LIN {X 91.341,Y 104.941,Z 79.000,A 180.000,B 0.000,C 180.000} C_DIS
LIN {X 91.355,Y 104.953,Z 79.000,A 180.000,B 0.000,C 180.000} C_DIS
LIN {X 91.533,Y 105.100,Z 79.000,A 180.000,B 0.000,C 180.000} C_DIS
LIN {X 91.560,Y 105.120,Z 79.000,A 180.000,B 0.000,C 180.000} C_DIS
LIN {X 91.712,Y 105.235,Z 79.000,A 180.000,B 0.000,C 180.000} C_DIS
LIN {X 91.797,Y 105.299,Z 79.000,A 180.000,B 0.000,C 180.000} C_DIS
LIN {X 91.891,Y 105.368,Z 79.000,A 180.000,B 0.000,C 180.000} C_DIS
LIN {X 92.052,Y 105.477,Z 79.000,A 180.000,B 0.000,C 180.000} C_DIS
LIN {X 92.070,Y 105.489,Z 79.000,A 180.000,B 0.000,C 180.000} C_DIS
LIN {X 92.249,Y 105.609,Z 79.000,A 180.000,B 0.000,C 180.000} C_DIS
LIN {X 92.323,Y 105.656,Z 79.000,A 180.000,B 0.000,C 180.000} C_DIS
LIN {X 92.427,Y 105.722,Z 79.000,A 180.000,B 0.000,C 180.000} C_DIS
LIN {X 92.606,Y 105.829,Z 79.000,A 180.000,B 0.000,C 180.000} C_DIS
LIN {X 92.785,Y 105.934,Z 79.000,A 180.000,B 0.000,C 180.000} C_DIS
LIN {X 92.933,Y 106.014,Z 79.000,A 180.000,B 0.000,C 180.000} C_DIS
LIN {X 93.142,Y 106.122,Z 79.000,A 180.000,B 0.000,C 180.000} C_DIS
LIN {X 93.284,Y 106.193,Z 79.000,A 180.000,B 0.000,C 180.000} C_DIS
LIN {X 93.321,Y 106.210,Z 79.000,A 180.000,B 0.000,C 180.000} C_DIS
LIN {X 93.500,Y 106.293,Z 79.000,A 180.000,B 0.000,C 180.000} C_DIS
LIN {X 93.679,Y 106.373,Z 79.000,A 180.000,B 0.000,C 180.000} C_DIS
LIN {X 93.857,Y 106.450,Z 79.000,A 180.000,B 0.000,C 180.000} C_DIS
LIN {X 94.036,Y 106.518,Z 79.000,A 180.000,B 0.000,C 180.000} C_DIS
LIN {X 94.119,Y 106.550,Z 79.000,A 180.000,B 0.000,C 180.000} C_DIS
LIN {X 94.215,Y 106.587,Z 79.000,A 180.000,B 0.000,C 180.000} C_DIS
LIN {X 94.321,Y 106.622,Z 79.000,A 180.000,B 0.000,C 180.000} C_DIS
; Link Move Starts
LIN {X 94.610,Y 106.716,Z 79.000,A 180.000,B 0.000,C 180.000} C_DIS
LIN {X 94.889,Y 106.804,Z 78.999,A 180.000,B 0.000,C 180.000} C_DIS
LIN {X 95.191,Y 106.882,Z 78.998,A 180.000,B 0.000,C 180.000} C_DIS
LIN {X 95.473,Y 106.946,Z 78.996,A 180.000,B 0.000,C 180.000} C_DIS
LIN {X 95.778,Y 107.008,Z 78.994,A 180.000,B 0.000,C 180.000} C_DIS
LIN {X 96.070,Y 107.058,Z 78.992,A 180.000,B 0.000,C 180.000} C_DIS
LIN {X 96.375,Y 107.102,Z 78.989,A 180.000,B 0.000,C 180.000} C_DIS
LIN {X 96.666,Y 107.130,Z 78.986,A 180.000,B 0.000,C 180.000} C_DIS
LIN {X 96.966,Y 107.154,Z 78.983,A 180.000,B 0.000,C 180.000} C_DIS
LIN {X 97.269,Y 107.168,Z 78.979,A 180.000,B 0.000,C 180.000} C_DIS
LIN {X 97.568,Y 107.174,Z 78.974,A 180.000,B 0.000,C 180.000} C_DIS
LIN {X 97.873,Y 107.168,Z 78.970,A 180.000,B 0.000,C 180.000} C_DIS
LIN {X 98.166,Y 107.154,Z 78.965,A 180.000,B 0.000,C 180.000} C_DIS
LIN {X 98.319,Y 107.143,Z 78.962,A 180.000,B 0.000,C 180.000} C_DIS
LIN {X 98.472,Y 107.131,Z 78.959,A 180.000,B 0.000,C 180.000} C_DIS
LIN {X 98.619,Y 107.118,Z 78.956,A 180.000,B 0.000,C 180.000} C_DIS
LIN {X 98.766,Y 107.100,Z 78.953,A 180.000,B 0.000,C 180.000} C_DIS
LIN {X 98.917,Y 107.080,Z 78.950,A 180.000,B 0.000,C 180.000} C_DIS
LIN {X 99.068,Y 107.059,Z 78.947,A 180.000,B 0.000,C 180.000} C_DIS
LIN {X 99.216,Y 107.033,Z 78.944,A 180.000,B 0.000,C 180.000} C_DIS
LIN {X 99.364,Y 107.005,Z 78.941,A 180.000,B 0.000,C 180.000} C_DIS
LIN {X 99.513,Y 106.977,Z 78.937,A 180.000,B 0.000,C 180.000} C_DIS
LIN {X 99.662,Y 106.949,Z 78.934,A 180.000,B 0.000,C 180.000} C_DIS
LIN {X 99.809,Y 106.915,Z 78.930,A 180.000,B 0.000,C 180.000} C_DIS
LIN {X 99.956,Y 106.879,Z 78.927,A 180.000,B 0.000,C 180.000} C_DIS
LIN {X 100.097,Y 106.844,Z 78.923,A 180.000,B 0.000,C 180.000} C_DIS
LIN {X 100.238,Y 106.804,Z 78.920,A 180.000,B 0.000,C 180.000} C_DIS
LIN {X 100.387,Y 106.758,Z 78.916,A 180.000,B 0.000,C 180.000} C_DIS
LIN {X 100.537,Y 106.713,Z 78.912,A 180.000,B 0.000,C 180.000} C_DIS
LIN {X 100.680,Y 106.668,Z 78.908,A 180.000,B 0.000,C 180.000} C_DIS
LIN {X 100.823,Y 106.620,Z 78.904,A 180.000,B 0.000,C 180.000} C_DIS
LIN {X 100.965,Y 106.568,Z 78.900,A 180.000,B 0.000,C 180.000} C_DIS
LIN {X 101.108,Y 106.516,Z 78.896,A 180.000,B 0.000,C 180.000} C_DIS
LIN {X 101.245,Y 106.462,Z 78.891,A 180.000,B 0.000,C 180.000} C_DIS
LIN {X 101.381,Y 106.403,Z 78.887,A 180.000,B 0.000,C 180.000} C_DIS
LIN {X 101.523,Y 106.342,Z 78.883,A 180.000,B 0.000,C 180.000} C_DIS
LIN {X 101.665,Y 106.279,Z 78.878,A 180.000,B 0.000,C 180.000} C_DIS
LIN {X 101.800,Y 106.218,Z 78.874,A 180.000,B 0.000,C 180.000} C_DIS
LIN {X 101.934,Y 106.151,Z 78.869,A 180.000,B 0.000,C 180.000} C_DIS
LIN {X 102.068,Y 106.084,Z 78.864,A 180.000,B 0.000,C 180.000} C_DIS
LIN {X 102.203,Y 106.016,Z 78.860,A 180.000,B 0.000,C 180.000} C_DIS
LIN {X 102.336,Y 105.941,Z 78.855,A 180.000,B 0.000,C 180.000} C_DIS
LIN {X 102.470,Y 105.865,Z 78.850,A 180.000,B 0.000,C 180.000} C_DIS
LIN {X 102.601,Y 105.790,Z 78.845,A 180.000,B 0.000,C 180.000} C_DIS
LIN {X 102.730,Y 105.711,Z 78.840,A 180.000,B 0.000,C 180.000} C_DIS
LIN {X 102.795,Y 105.671,Z 78.838,A 180.000,B 0.000,C 180.000} C_DIS
LIN {X 102.859,Y 105.629,Z 78.835,A 180.000,B 0.000,C 180.000} C_DIS
LIN {X 102.923,Y 105.588,Z 78.833,A 180.000,B 0.000,C 180.000} C_DIS
LIN {X 102.987,Y 105.546,Z 78.830,A 180.000,B 0.000,C 180.000} C_DIS
LIN {X 103.050,Y 105.506,Z 78.828,A 180.000,B 0.000,C 180.000} C_DIS
LIN {X 103.113,Y 105.465,Z 78.825,A 180.000,B 0.000,C 180.000} C_DIS
LIN {X 103.174,Y 105.423,Z 78.823,A 180.000,B 0.000,C 180.000} C_DIS
LIN {X 103.235,Y 105.380,Z 78.820,A 180.000,B 0.000,C 180.000} C_DIS
LIN {X 103.298,Y 105.334,Z 78.817,A 180.000,B 0.000,C 180.000} C_DIS
LIN {X 103.422,Y 105.243,Z 78.812,A 180.000,B 0.000,C 180.000} C_DIS
LIN {X 103.485,Y 105.198,Z 78.809,A 180.000,B 0.000,C 180.000} C_DIS
LIN {X 103.544,Y 105.153,Z 78.807,A 180.000,B 0.000,C 180.000} C_DIS
LIN {X 103.602,Y 105.107,Z 78.804,A 180.000,B 0.000,C 180.000} C_DIS
LIN {X 103.659,Y 105.061,Z 78.802,A 180.000,B 0.000,C 180.000} C_DIS
LIN {X 103.717,Y 105.015,Z 78.799,A 180.000,B 0.000,C 180.000} C_DIS
LIN {X 103.839,Y 104.915,Z 78.793,A 180.000,B 0.000,C 180.000} C_DIS
LIN {X 103.960,Y 104.816,Z 78.788,A 180.000,B 0.000,C 180.000} C_DIS
LIN {X 104.017,Y 104.769,Z 78.785,A 180.000,B 0.000,C 180.000} C_DIS
LIN {X 104.073,Y 104.720,Z 78.783,A 180.000,B 0.000,C 180.000} C_DIS
LIN {X 104.127,Y 104.671,Z 78.780,A 180.000,B 0.000,C 180.000} C_DIS
LIN {X 104.181,Y 104.621,Z 78.778,A 180.000,B 0.000,C 180.000} C_DIS
LIN {X 104.293,Y 104.519,Z 78.772,A 180.000,B 0.000,C 180.000} C_DIS
LIN {X 104.348,Y 104.468,Z 78.770,A 180.000,B 0.000,C 180.000} C_DIS
LIN {X 104.402,Y 104.416,Z 78.767,A 180.000,B 0.000,C 180.000} C_DIS
LIN {X 104.456,Y 104.361,Z 78.764,A 180.000,B 0.000,C 180.000} C_DIS
LIN {X 104.564,Y 104.250,Z 78.759,A 180.000,B 0.000,C 180.000} C_DIS
LIN {X 104.618,Y 104.195,Z 78.756,A 180.000,B 0.000,C 180.000} C_DIS
LIN {X 104.671,Y 104.141,Z 78.754,A 180.000,B 0.000,C 180.000} C_DIS
LIN {X 104.776,Y 104.032,Z 78.748,A 180.000,B 0.000,C 180.000} C_DIS
LIN {X 104.828,Y 103.978,Z 78.746,A 180.000,B 0.000,C 180.000} C_DIS
LIN {X 104.880,Y 103.920,Z 78.743,A 180.000,B 0.000,C 180.000} C_DIS
LIN {X 104.981,Y 103.804,Z 78.738,A 180.000,B 0.000,C 180.000} C_DIS
LIN {X 105.032,Y 103.746,Z 78.735,A 180.000,B 0.000,C 180.000} C_DIS
LIN {X 105.080,Y 103.690,Z 78.732,A 180.000,B 0.000,C 180.000} C_DIS
LIN {X 105.129,Y 103.634,Z 78.730,A 180.000,B 0.000,C 180.000} C_DIS
LIN {X 105.175,Y 103.577,Z 78.727,A 180.000,B 0.000,C 180.000} C_DIS
LIN {X 105.221,Y 103.518,Z 78.725,A 180.000,B 0.000,C 180.000} C_DIS
LIN {X 105.316,Y 103.396,Z 78.719,A 180.000,B 0.000,C 180.000} C_DIS
LIN {X 105.364,Y 103.334,Z 78.717,A 180.000,B 0.000,C 180.000} C_DIS
LIN {X 105.411,Y 103.273,Z 78.714,A 180.000,B 0.000,C 180.000} C_DIS
LIN {X 105.502,Y 103.153,Z 78.709,A 180.000,B 0.000,C 180.000} C_DIS
LIN {X 105.546,Y 103.092,Z 78.706,A 180.000,B 0.000,C 180.000} C_DIS
LIN {X 105.590,Y 103.030,Z 78.703,A 180.000,B 0.000,C 180.000} C_DIS
LIN {X 105.676,Y 102.905,Z 78.698,A 180.000,B 0.000,C 180.000} C_DIS
LIN {X 105.763,Y 102.779,Z 78.693,A 180.000,B 0.000,C 180.000} C_DIS
LIN {X 105.806,Y 102.715,Z 78.690,A 180.000,B 0.000,C 180.000} C_DIS
LIN {X 105.847,Y 102.650,Z 78.687,A 180.000,B 0.000,C 180.000} C_DIS
LIN {X 106.006,Y 102.389,Z 78.677,A 180.000,B 0.000,C 180.000} C_DIS
LIN {X 106.046,Y 102.324,Z 78.674,A 180.000,B 0.000,C 180.000} C_DIS
LIN {X 106.084,Y 102.257,Z 78.671,A 180.000,B 0.000,C 180.000} C_DIS
LIN {X 106.122,Y 102.191,Z 78.669,A 180.000,B 0.000,C 180.000} C_DIS
LIN {X 106.159,Y 102.124,Z 78.666,A 180.000,B 0.000,C 180.000} C_DIS
LIN {X 106.196,Y 102.056,Z 78.663,A 180.000,B 0.000,C 180.000} C_DIS
LIN {X 106.268,Y 101.922,Z 78.658,A 180.000,B 0.000,C 180.000} C_DIS
LIN {X 106.303,Y 101.856,Z 78.655,A 180.000,B 0.000,C 180.000} C_DIS
LIN {X 106.339,Y 101.790,Z 78.653,A 180.000,B 0.000,C 180.000} C_DIS
LIN {X 106.372,Y 101.723,Z 78.650,A 180.000,B 0.000,C 180.000} C_DIS
LIN {X 106.406,Y 101.652,Z 78.647,A 180.000,B 0.000,C 180.000} C_DIS
LIN {X 106.505,Y 101.440,Z 78.639,A 180.000,B 0.000,C 180.000} C_DIS
LIN {X 106.537,Y 101.371,Z 78.637,A 180.000,B 0.000,C 180.000} C_DIS
LIN {X 106.567,Y 101.302,Z 78.634,A 180.000,B 0.000,C 180.000} C_DIS
LIN {X 106.597,Y 101.232,Z 78.631,A 180.000,B 0.000,C 180.000} C_DIS
LIN {X 106.625,Y 101.163,Z 78.629,A 180.000,B 0.000,C 180.000} C_DIS
LIN {X 106.655,Y 101.091,Z 78.626,A 180.000,B 0.000,C 180.000} C_DIS
LIN {X 106.769,Y 100.805,Z 78.615,A 180.000,B 0.000,C 180.000} C_DIS
LIN {X 106.797,Y 100.735,Z 78.613,A 180.000,B 0.000,C 180.000} C_DIS
LIN {X 106.822,Y 100.664,Z 78.610,A 180.000,B 0.000,C 180.000} C_DIS
LIN {X 106.846,Y 100.593,Z 78.607,A 180.000,B 0.000,C 180.000} C_DIS
LIN {X 106.920,Y 100.372,Z 78.599,A 180.000,B 0.000,C 180.000} C_DIS
LIN {X 106.945,Y 100.299,Z 78.596,A 180.000,B 0.000,C 180.000} C_DIS
LIN {X 106.967,Y 100.226,Z 78.594,A 180.000,B 0.000,C 180.000} C_DIS
LIN {X 106.987,Y 100.153,Z 78.591,A 180.000,B 0.000,C 180.000} C_DIS
LIN {X 107.048,Y 99.930,Z 78.583,A 180.000,B 0.000,C 180.000} C_DIS
LIN {X 107.069,Y 99.855,Z 78.580,A 180.000,B 0.000,C 180.000} C_DIS
LIN {X 107.090,Y 99.779,Z 78.578,A 180.000,B 0.000,C 180.000} C_DIS
LIN {X 107.111,Y 99.703,Z 78.575,A 180.000,B 0.000,C 180.000} C_DIS
LIN {X 107.129,Y 99.630,Z 78.572,A 180.000,B 0.000,C 180.000} C_DIS
LIN {X 107.145,Y 99.557,Z 78.570,A 180.000,B 0.000,C 180.000} C_DIS
LIN {X 107.209,Y 99.262,Z 78.559,A 180.000,B 0.000,C 180.000} C_DIS
LIN {X 107.224,Y 99.188,Z 78.556,A 180.000,B 0.000,C 180.000} C_DIS
LIN {X 107.237,Y 99.114,Z 78.554,A 180.000,B 0.000,C 180.000} C_DIS
LIN {X 107.286,Y 98.806,Z 78.543,A 180.000,B 0.000,C 180.000} C_DIS
LIN {X 107.298,Y 98.729,Z 78.540,A 180.000,B 0.000,C 180.000} C_DIS
LIN {X 107.320,Y 98.575,Z 78.535,A 180.000,B 0.000,C 180.000} C_DIS
LIN {X 107.329,Y 98.498,Z 78.532,A 180.000,B 0.000,C 180.000} C_DIS
LIN {X 107.337,Y 98.422,Z 78.529,A 180.000,B 0.000,C 180.000} C_DIS
LIN {X 107.360,Y 98.192,Z 78.521,A 180.000,B 0.000,C 180.000} C_DIS
LIN {X 107.368,Y 98.117,Z 78.519,A 180.000,B 0.000,C 180.000} C_DIS
LIN {X 107.374,Y 98.042,Z 78.516,A 180.000,B 0.000,C 180.000} C_DIS
LIN {X 107.378,Y 97.967,Z 78.513,A 180.000,B 0.000,C 180.000} C_DIS
LIN {X 107.391,Y 97.660,Z 78.503,A 180.000,B 0.000,C 180.000} C_DIS
LIN {X 107.394,Y 97.583,Z 78.500,A 180.000,B 0.000,C 180.000} C_DIS
LIN {X 107.396,Y 97.429,Z 78.495,A 180.000,B 0.000,C 180.000} C_DIS
LIN {X 107.397,Y 97.352,Z 78.492,A 180.000,B 0.000,C 180.000} C_DIS
LIN {X 107.393,Y 97.040,Z 78.481,A 180.000,B 0.000,C 180.000} C_DIS
LIN {X 107.392,Y 96.962,Z 78.478,A 180.000,B 0.000,C 180.000} C_DIS
LIN {X 107.388,Y 96.886,Z 78.476,A 180.000,B 0.000,C 180.000} C_DIS
LIN {X 107.383,Y 96.810,Z 78.473,A 180.000,B 0.000,C 180.000} C_DIS
LIN {X 107.368,Y 96.581,Z 78.465,A 180.000,B 0.000,C 180.000} C_DIS
LIN {X 107.362,Y 96.505,Z 78.462,A 180.000,B 0.000,C 180.000} C_DIS
LIN {X 107.355,Y 96.429,Z 78.460,A 180.000,B 0.000,C 180.000} C_DIS
LIN {X 107.347,Y 96.353,Z 78.457,A 180.000,B 0.000,C 180.000} C_DIS
LIN {X 107.339,Y 96.275,Z 78.454,A 180.000,B 0.000,C 180.000} C_DIS
LIN {X 107.329,Y 96.198,Z 78.452,A 180.000,B 0.000,C 180.000} C_DIS
LIN {X 107.291,Y 95.890,Z 78.441,A 180.000,B 0.000,C 180.000} C_DIS
LIN {X 107.281,Y 95.814,Z 78.438,A 180.000,B 0.000,C 180.000} C_DIS
LIN {X 107.268,Y 95.739,Z 78.435,A 180.000,B 0.000,C 180.000} C_DIS
LIN {X 107.212,Y 95.433,Z 78.425,A 180.000,B 0.000,C 180.000} C_DIS
LIN {X 107.198,Y 95.358,Z 78.422,A 180.000,B 0.000,C 180.000} C_DIS
LIN {X 107.182,Y 95.283,Z 78.419,A 180.000,B 0.000,C 180.000} C_DIS
LIN {X 107.164,Y 95.209,Z 78.417,A 180.000,B 0.000,C 180.000} C_DIS
LIN {X 107.147,Y 95.135,Z 78.414,A 180.000,B 0.000,C 180.000} C_DIS
LIN {X 107.128,Y 95.058,Z 78.411,A 180.000,B 0.000,C 180.000} C_DIS
LIN {X 107.073,Y 94.828,Z 78.403,A 180.000,B 0.000,C 180.000} C_DIS
LIN {X 107.055,Y 94.754,Z 78.400,A 180.000,B 0.000,C 180.000} C_DIS
LIN {X 107.035,Y 94.681,Z 78.398,A 180.000,B 0.000,C 180.000} C_DIS
LIN {X 107.014,Y 94.608,Z 78.395,A 180.000,B 0.000,C 180.000} C_DIS
LIN {X 106.970,Y 94.461,Z 78.390,A 180.000,B 0.000,C 180.000} C_DIS
LIN {X 106.925,Y 94.314,Z 78.384,A 180.000,B 0.000,C 180.000} C_DIS
LIN {X 106.902,Y 94.241,Z 78.381,A 180.000,B 0.000,C 180.000} C_DIS
LIN {X 106.877,Y 94.167,Z 78.379,A 180.000,B 0.000,C 180.000} C_DIS
LIN {X 106.770,Y 93.873,Z 78.368,A 180.000,B 0.000,C 180.000} C_DIS
LIN {X 106.743,Y 93.800,Z 78.365,A 180.000,B 0.000,C 180.000} C_DIS
LIN {X 106.716,Y 93.728,Z 78.362,A 180.000,B 0.000,C 180.000} C_DIS
LIN {X 106.688,Y 93.655,Z 78.360,A 180.000,B 0.000,C 180.000} C_DIS
LIN {X 106.659,Y 93.583,Z 78.357,A 180.000,B 0.000,C 180.000} C_DIS
LIN {X 106.629,Y 93.512,Z 78.354,A 180.000,B 0.000,C 180.000} C_DIS
LIN {X 106.538,Y 93.299,Z 78.346,A 180.000,B 0.000,C 180.000} C_DIS
LIN {X 106.507,Y 93.228,Z 78.343,A 180.000,B 0.000,C 180.000} C_DIS
LIN {X 106.475,Y 93.158,Z 78.341,A 180.000,B 0.000,C 180.000} C_DIS
LIN {X 106.441,Y 93.089,Z 78.338,A 180.000,B 0.000,C 180.000} C_DIS
LIN {X 106.372,Y 92.949,Z 78.333,A 180.000,B 0.000,C 180.000} C_DIS
LIN {X 106.303,Y 92.810,Z 78.327,A 180.000,B 0.000,C 180.000} C_DIS
LIN {X 106.267,Y 92.741,Z 78.325,A 180.000,B 0.000,C 180.000} C_DIS
LIN {X 106.231,Y 92.672,Z 78.322,A 180.000,B 0.000,C 180.000} C_DIS
LIN {X 106.194,Y 92.603,Z 78.319,A 180.000,B 0.000,C 180.000} C_DIS
LIN {X 106.157,Y 92.535,Z 78.316,A 180.000,B 0.000,C 180.000} C_DIS
LIN {X 106.080,Y 92.400,Z 78.311,A 180.000,B 0.000,C 180.000} C_DIS
LIN {X 106.003,Y 92.265,Z 78.306,A 180.000,B 0.000,C 180.000} C_DIS
LIN {X 105.965,Y 92.198,Z 78.303,A 180.000,B 0.000,C 180.000} C_DIS
LIN {X 105.924,Y 92.132,Z 78.300,A 180.000,B 0.000,C 180.000} C_DIS
LIN {X 105.882,Y 92.067,Z 78.297,A 180.000,B 0.000,C 180.000} C_DIS
LIN {X 105.840,Y 92.002,Z 78.295,A 180.000,B 0.000,C 180.000} C_DIS
LIN {X 105.756,Y 91.872,Z 78.289,A 180.000,B 0.000,C 180.000} C_DIS
LIN {X 105.714,Y 91.807,Z 78.287,A 180.000,B 0.000,C 180.000} C_DIS
LIN {X 105.670,Y 91.743,Z 78.284,A 180.000,B 0.000,C 180.000} C_DIS
LIN {X 105.581,Y 91.615,Z 78.278,A 180.000,B 0.000,C 180.000} C_DIS
LIN {X 105.535,Y 91.551,Z 78.276,A 180.000,B 0.000,C 180.000} C_DIS
LIN {X 105.489,Y 91.488,Z 78.273,A 180.000,B 0.000,C 180.000} C_DIS
LIN {X 105.398,Y 91.363,Z 78.268,A 180.000,B 0.000,C 180.000} C_DIS
LIN {X 105.353,Y 91.301,Z 78.265,A 180.000,B 0.000,C 180.000} C_DIS
LIN {X 105.306,Y 91.239,Z 78.262,A 180.000,B 0.000,C 180.000} C_DIS
LIN {X 105.257,Y 91.177,Z 78.259,A 180.000,B 0.000,C 180.000} C_DIS
LIN {X 105.158,Y 91.056,Z 78.254,A 180.000,B 0.000,C 180.000} C_DIS
LIN {X 105.108,Y 90.995,Z 78.251,A 180.000,B 0.000,C 180.000} C_DIS
LIN {X 105.059,Y 90.935,Z 78.249,A 180.000,B 0.000,C 180.000} C_DIS
LIN {X 105.009,Y 90.875,Z 78.246,A 180.000,B 0.000,C 180.000} C_DIS
LIN {X 104.958,Y 90.817,Z 78.243,A 180.000,B 0.000,C 180.000} C_DIS
LIN {X 104.906,Y 90.760,Z 78.240,A 180.000,B 0.000,C 180.000} C_DIS
LIN {X 104.853,Y 90.702,Z 78.238,A 180.000,B 0.000,C 180.000} C_DIS
LIN {X 104.800,Y 90.644,Z 78.235,A 180.000,B 0.000,C 180.000} C_DIS
LIN {X 104.642,Y 90.471,Z 78.227,A 180.000,B 0.000,C 180.000} C_DIS
LIN {X 104.590,Y 90.414,Z 78.224,A 180.000,B 0.000,C 180.000} C_DIS
LIN {X 104.536,Y 90.358,Z 78.221,A 180.000,B 0.000,C 180.000} C_DIS
LIN {X 104.481,Y 90.304,Z 78.219,A 180.000,B 0.000,C 180.000} C_DIS
LIN {X 104.369,Y 90.195,Z 78.213,A 180.000,B 0.000,C 180.000} C_DIS
LIN {X 104.257,Y 90.085,Z 78.208,A 180.000,B 0.000,C 180.000} C_DIS
LIN {X 104.200,Y 90.032,Z 78.205,A 180.000,B 0.000,C 180.000} C_DIS
LIN {X 104.142,Y 89.980,Z 78.202,A 180.000,B 0.000,C 180.000} C_DIS
LIN {X 103.966,Y 89.826,Z 78.194,A 180.000,B 0.000,C 180.000} C_DIS
LIN {X 103.906,Y 89.774,Z 78.191,A 180.000,B 0.000,C 180.000} C_DIS
LIN {X 103.847,Y 89.723,Z 78.189,A 180.000,B 0.000,C 180.000} C_DIS
LIN {X 103.787,Y 89.672,Z 78.186,A 180.000,B 0.000,C 180.000} C_DIS
LIN {X 103.728,Y 89.622,Z 78.183,A 180.000,B 0.000,C 180.000} C_DIS
LIN {X 103.667,Y 89.573,Z 78.181,A 180.000,B 0.000,C 180.000} C_DIS
LIN {X 103.606,Y 89.525,Z 78.178,A 180.000,B 0.000,C 180.000} C_DIS
LIN {X 103.483,Y 89.429,Z 78.173,A 180.000,B 0.000,C 180.000} C_DIS
LIN {X 103.421,Y 89.381,Z 78.170,A 180.000,B 0.000,C 180.000} C_DIS
LIN {X 103.358,Y 89.333,Z 78.167,A 180.000,B 0.000,C 180.000} C_DIS
LIN {X 103.295,Y 89.286,Z 78.165,A 180.000,B 0.000,C 180.000} C_DIS
LIN {X 103.231,Y 89.242,Z 78.162,A 180.000,B 0.000,C 180.000} C_DIS
LIN {X 103.167,Y 89.198,Z 78.160,A 180.000,B 0.000,C 180.000} C_DIS
LIN {X 103.103,Y 89.153,Z 78.157,A 180.000,B 0.000,C 180.000} C_DIS
LIN {X 103.039,Y 89.109,Z 78.155,A 180.000,B 0.000,C 180.000} C_DIS
LIN {X 102.974,Y 89.065,Z 78.152,A 180.000,B 0.000,C 180.000} C_DIS
LIN {X 102.909,Y 89.021,Z 78.150,A 180.000,B 0.000,C 180.000} C_DIS
LIN {X 102.778,Y 88.935,Z 78.145,A 180.000,B 0.000,C 180.000} C_DIS
LIN {X 102.644,Y 88.854,Z 78.140,A 180.000,B 0.000,C 180.000} C_DIS
LIN {X 102.511,Y 88.772,Z 78.135,A 180.000,B 0.000,C 180.000} C_DIS
LIN {X 102.377,Y 88.691,Z 78.130,A 180.000,B 0.000,C 180.000} C_DIS
LIN {X 102.240,Y 88.617,Z 78.126,A 180.000,B 0.000,C 180.000} C_DIS
LIN {X 102.102,Y 88.543,Z 78.121,A 180.000,B 0.000,C 180.000} C_DIS
LIN {X 101.963,Y 88.469,Z 78.116,A 180.000,B 0.000,C 180.000} C_DIS
LIN {X 101.823,Y 88.400,Z 78.112,A 180.000,B 0.000,C 180.000} C_DIS
LIN {X 101.681,Y 88.333,Z 78.108,A 180.000,B 0.000,C 180.000} C_DIS
LIN {X 101.539,Y 88.267,Z 78.103,A 180.000,B 0.000,C 180.000} C_DIS
LIN {X 101.396,Y 88.201,Z 78.099,A 180.000,B 0.000,C 180.000} C_DIS
LIN {X 101.252,Y 88.140,Z 78.095,A 180.000,B 0.000,C 180.000} C_DIS
LIN {X 101.106,Y 88.082,Z 78.091,A 180.000,B 0.000,C 180.000} C_DIS
LIN {X 100.961,Y 88.025,Z 78.087,A 180.000,B 0.000,C 180.000} C_DIS
LIN {X 100.814,Y 87.971,Z 78.083,A 180.000,B 0.000,C 180.000} C_DIS
LIN {X 100.664,Y 87.920,Z 78.079,A 180.000,B 0.000,C 180.000} C_DIS
LIN {X 100.515,Y 87.871,Z 78.075,A 180.000,B 0.000,C 180.000} C_DIS
LIN {X 100.366,Y 87.822,Z 78.071,A 180.000,B 0.000,C 180.000} C_DIS
LIN {X 100.216,Y 87.775,Z 78.067,A 180.000,B 0.000,C 180.000} C_DIS
LIN {X 100.065,Y 87.734,Z 78.064,A 180.000,B 0.000,C 180.000} C_DIS
LIN {X 99.913,Y 87.693,Z 78.060,A 180.000,B 0.000,C 180.000} C_DIS
LIN {X 99.761,Y 87.654,Z 78.057,A 180.000,B 0.000,C 180.000} C_DIS
LIN {X 99.607,Y 87.621,Z 78.054,A 180.000,B 0.000,C 180.000} C_DIS
LIN {X 99.453,Y 87.589,Z 78.050,A 180.000,B 0.000,C 180.000} C_DIS
LIN {X 99.299,Y 87.557,Z 78.047,A 180.000,B 0.000,C 180.000} C_DIS
LIN {X 99.145,Y 87.527,Z 78.044,A 180.000,B 0.000,C 180.000} C_DIS
LIN {X 98.990,Y 87.503,Z 78.041,A 180.000,B 0.000,C 180.000} C_DIS
LIN {X 98.834,Y 87.479,Z 78.038,A 180.000,B 0.000,C 180.000} C_DIS
LIN {X 98.679,Y 87.456,Z 78.036,A 180.000,B 0.000,C 180.000} C_DIS
LIN {X 98.522,Y 87.440,Z 78.033,A 180.000,B 0.000,C 180.000} C_DIS
LIN {X 98.365,Y 87.425,Z 78.030,A 180.000,B 0.000,C 180.000} C_DIS
LIN {X 98.052,Y 87.400,Z 78.026,A 180.000,B 0.000,C 180.000} C_DIS
LIN {X 97.737,Y 87.386,Z 78.021,A 180.000,B 0.000,C 180.000} C_DIS
LIN {X 97.423,Y 87.380,Z 78.017,A 180.000,B 0.000,C 180.000} C_DIS
LIN {X 97.108,Y 87.387,Z 78.013,A 180.000,B 0.000,C 180.000} C_DIS
LIN {X 96.793,Y 87.403,Z 78.010,A 180.000,B 0.000,C 180.000} C_DIS
LIN {X 96.479,Y 87.428,Z 78.007,A 180.000,B 0.000,C 180.000} C_DIS
LIN {X 96.167,Y 87.463,Z 78.005,A 180.000,B 0.000,C 180.000} C_DIS
LIN {X 95.855,Y 87.508,Z 78.003,A 180.000,B 0.000,C 180.000} C_DIS
LIN {X 95.545,Y 87.566,Z 78.002,A 180.000,B 0.000,C 180.000} C_DIS
LIN {X 95.236,Y 87.628,Z 78.001,A 180.000,B 0.000,C 180.000} C_DIS
LIN {X 94.931,Y 87.704,Z 78.000,A 180.000,B 0.000,C 180.000} C_DIS
LIN {X 94.776,Y 87.747,Z 78.000,A 180.000,B 0.000,C 180.000} C_DIS
; Cutting Move Starts
LIN {X 94.751,Y 87.754,Z 78.000,A 180.000,B 0.000,C 180.000} C_DIS
LIN {X 94.665,Y 87.779,Z 78.000,A 180.000,B 0.000,C 180.000} C_DIS
LIN {X 94.394,Y 87.866,Z 78.000,A 180.000,B 0.000,C 180.000} C_DIS
LIN {X 94.215,Y 87.923,Z 78.000,A 180.000,B 0.000,C 180.000} C_DIS
LIN {X 94.110,Y 87.958,Z 78.000,A 180.000,B 0.000,C 180.000} C_DIS
LIN {X 94.036,Y 87.985,Z 78.000,A 180.000,B 0.000,C 180.000} C_DIS
LIN {X 93.857,Y 88.053,Z 78.000,A 180.000,B 0.000,C 180.000} C_DIS
LIN {X 93.679,Y 88.122,Z 78.000,A 180.000,B 0.000,C 180.000} C_DIS
LIN {X 93.642,Y 88.137,Z 78.000,A 180.000,B 0.000,C 180.000} C_DIS
LIN {X 93.500,Y 88.199,Z 78.000,A 180.000,B 0.000,C 180.000} C_DIS
LIN {X 93.321,Y 88.279,Z 78.000,A 180.000,B 0.000,C 180.000} C_DIS
LIN {X 93.240,Y 88.316,Z 78.000,A 180.000,B 0.000,C 180.000} C_DIS
LIN {X 93.142,Y 88.361,Z 78.000,A 180.000,B 0.000,C 180.000} C_DIS
LIN {X 92.964,Y 88.448,Z 78.000,A 180.000,B 0.000,C 180.000} C_DIS
LIN {X 92.785,Y 88.541,Z 78.000,A 180.000,B 0.000,C 180.000} C_DIS
LIN {X 92.606,Y 88.634,Z 78.000,A 180.000,B 0.000,C 180.000} C_DIS
LIN {X 92.538,Y 88.673,Z 78.000,A 180.000,B 0.000,C 180.000} C_DIS
LIN {X 92.235,Y 88.852,Z 78.000,A 180.000,B 0.000,C 180.000} C_DIS
LIN {X 92.070,Y 88.955,Z 78.000,A 180.000,B 0.000,C 180.000} C_DIS
LIN {X 91.953,Y 89.031,Z 78.000,A 180.000,B 0.000,C 180.000} C_DIS
LIN {X 91.686,Y 89.209,Z 78.000,A 180.000,B 0.000,C 180.000} C_DIS
LIN {X 91.533,Y 89.319,Z 78.000,A 180.000,B 0.000,C 180.000} C_DIS
LIN {X 91.355,Y 89.454,Z 78.000,A 180.000,B 0.000,C 180.000} C_DIS
LIN {X 91.207,Y 89.567,Z 78.000,A 180.000,B 0.000,C 180.000} C_DIS
LIN {X 91.176,Y 89.593,Z 78.000,A 180.000,B 0.000,C 180.000} C_DIS
LIN {X 90.997,Y 89.742,Z 78.000,A 180.000,B 0.000,C 180.000} C_DIS
LIN {X 90.781,Y 89.925,Z 78.000,A 180.000,B 0.000,C 180.000} C_DIS
LIN {X 90.640,Y 90.053,Z 78.000,A 180.000,B 0.000,C 180.000} C_DIS
LIN {X 90.461,Y 90.222,Z 78.000,A 180.000,B 0.000,C 180.000} C_DIS
LIN {X 90.398,Y 90.282,Z 78.000,A 180.000,B 0.000,C 180.000} C_DIS
LIN {X 90.282,Y 90.400,Z 78.000,A 180.000,B 0.000,C 180.000} C_DIS
LIN {X 90.103,Y 90.590,Z 78.000,A 180.000,B 0.000,C 180.000} C_DIS
LIN {X 90.056,Y 90.640,Z 78.000,A 180.000,B 0.000,C 180.000} C_DIS
LIN {X 89.925,Y 90.780,Z 78.000,A 180.000,B 0.000,C 180.000} C_DIS
LIN {X 89.891,Y 90.818,Z 78.000,A 180.000,B 0.000,C 180.000} C_DIS
LIN {X 89.746,Y 90.990,Z 78.000,A 180.000,B 0.000,C 180.000} C_DIS
LIN {X 89.740,Y 90.997,Z 78.000,A 180.000,B 0.000,C 180.000} C_DIS
LIN {X 89.591,Y 91.176,Z 78.000,A 180.000,B 0.000,C 180.000} C_DIS
LIN {X 89.567,Y 91.206,Z 78.000,A 180.000,B 0.000,C 180.000} C_DIS
LIN {X 89.455,Y 91.355,Z 78.000,A 180.000,B 0.000,C 180.000} C_DIS
LIN {X 89.388,Y 91.444,Z 78.000,A 180.000,B 0.000,C 180.000} C_DIS
LIN {X 89.321,Y 91.533,Z 78.000,A 180.000,B 0.000,C 180.000} C_DIS
LIN {X 89.209,Y 91.687,Z 78.000,A 180.000,B 0.000,C 180.000} C_DIS
LIN {X 89.192,Y 91.712,Z 78.000,A 180.000,B 0.000,C 180.000} C_DIS
LIN {X 89.072,Y 91.891,Z 78.000,A 180.000,B 0.000,C 180.000} C_DIS
LIN {X 89.031,Y 91.952,Z 78.000,A 180.000,B 0.000,C 180.000} C_DIS
LIN {X 88.952,Y 92.070,Z 78.000,A 180.000,B 0.000,C 180.000} C_DIS
LIN {X 88.852,Y 92.235,Z 78.000,A 180.000,B 0.000,C 180.000} C_DIS
LIN {X 88.738,Y 92.427,Z 78.000,A 180.000,B 0.000,C 180.000} C_DIS
LIN {X 88.673,Y 92.540,Z 78.000,A 180.000,B 0.000,C 180.000} C_DIS
LIN {X 88.637,Y 92.606,Z 78.000,A 180.000,B 0.000,C 180.000} C_DIS
LIN {X 88.541,Y 92.785,Z 78.000,A 180.000,B 0.000,C 180.000} C_DIS
LIN {X 88.449,Y 92.964,Z 78.000,A 180.000,B 0.000,C 180.000} C_DIS
LIN {X 88.359,Y 93.142,Z 78.000,A 180.000,B 0.000,C 180.000} C_DIS
LIN {X 88.316,Y 93.238,Z 78.000,A 180.000,B 0.000,C 180.000} C_DIS
LIN {X 88.198,Y 93.500,Z 78.000,A 180.000,B 0.000,C 180.000} C_DIS
LIN {X 88.137,Y 93.648,Z 78.000,A 180.000,B 0.000,C 180.000} C_DIS
LIN {X 88.124,Y 93.679,Z 78.000,A 180.000,B 0.000,C 180.000} C_DIS
LIN {X 88.055,Y 93.857,Z 78.000,A 180.000,B 0.000,C 180.000} C_DIS
LIN {X 87.958,Y 94.111,Z 78.000,A 180.000,B 0.000,C 180.000} C_DIS
LIN {X 87.921,Y 94.215,Z 78.000,A 180.000,B 0.000,C 180.000} C_DIS
LIN {X 87.864,Y 94.394,Z 78.000,A 180.000,B 0.000,C 180.000} C_DIS
LIN {X 87.807,Y 94.573,Z 78.000,A 180.000,B 0.000,C 180.000} C_DIS
LIN {X 87.779,Y 94.662,Z 78.000,A 180.000,B 0.000,C 180.000} C_DIS
LIN {X 87.755,Y 94.751,Z 78.000,A 180.000,B 0.000,C 180.000} C_DIS
LIN {X 87.709,Y 94.930,Z 78.000,A 180.000,B 0.000,C 180.000} C_DIS
LIN {X 87.663,Y 95.109,Z 78.000,A 180.000,B 0.000,C 180.000} C_DIS
LIN {X 87.618,Y 95.288,Z 78.000,A 180.000,B 0.000,C 180.000} C_DIS
LIN {X 87.601,Y 95.372,Z 78.000,A 180.000,B 0.000,C 180.000} C_DIS
LIN {X 87.546,Y 95.645,Z 78.000,A 180.000,B 0.000,C 180.000} C_DIS
LIN {X 87.513,Y 95.824,Z 78.000,A 180.000,B 0.000,C 180.000} C_DIS
LIN {X 87.488,Y 96.003,Z 78.000,A 180.000,B 0.000,C 180.000} C_DIS
LIN {X 87.463,Y 96.181,Z 78.000,A 180.000,B 0.000,C 180.000} C_DIS
LIN {X 87.442,Y 96.338,Z 78.000,A 180.000,B 0.000,C 180.000} C_DIS
LIN {X 87.439,Y 96.360,Z 78.000,A 180.000,B 0.000,C 180.000} C_DIS
LIN {X 87.422,Y 96.529,Z 78.000,A 180.000,B 0.000,C 180.000} C_DIS
LIN {X 87.406,Y 96.718,Z 78.000,A 180.000,B 0.000,C 180.000} C_DIS
LIN {X 87.391,Y 96.897,Z 78.000,A 180.000,B 0.000,C 180.000} C_DIS
LIN {X 87.384,Y 97.075,Z 78.000,A 180.000,B 0.000,C 180.000} C_DIS
LIN {X 87.379,Y 97.254,Z 78.000,A 180.000,B 0.000,C 180.000} C_DIS
LIN {X 87.375,Y 97.433,Z 78.000,A 180.000,B 0.000,C 180.000} C_DIS
LIN {X 87.376,Y 97.612,Z 78.000,A 180.000,B 0.000,C 180.000} C_DIS
LIN {X 87.380,Y 97.790,Z 78.000,A 180.000,B 0.000,C 180.000} C_DIS
LIN {X 87.385,Y 97.969,Z 78.000,A 180.000,B 0.000,C 180.000} C_DIS
LIN {X 87.394,Y 98.148,Z 78.000,A 180.000,B 0.000,C 180.000} C_DIS
LIN {X 87.425,Y 98.505,Z 78.000,A 180.000,B 0.000,C 180.000} C_DIS
LIN {X 87.445,Y 98.684,Z 78.000,A 180.000,B 0.000,C 180.000} C_DIS
LIN {X 87.469,Y 98.863,Z 78.000,A 180.000,B 0.000,C 180.000} C_DIS
LIN {X 87.494,Y 99.042,Z 78.000,A 180.000,B 0.000,C 180.000} C_DIS
LIN {X 87.520,Y 99.221,Z 78.000,A 180.000,B 0.000,C 180.000} C_DIS
LIN {X 87.555,Y 99.399,Z 78.000,A 180.000,B 0.000,C 180.000} C_DIS
LIN {X 87.601,Y 99.628,Z 78.000,A 180.000,B 0.000,C 180.000} C_DIS
LIN {X 87.629,Y 99.757,Z 78.000,A 180.000,B 0.000,C 180.000} C_DIS
LIN {X 87.675,Y 99.936,Z 78.000,A 180.000,B 0.000,C 180.000} C_DIS
LIN {X 87.721,Y 100.114,Z 78.000,A 180.000,B 0.000,C 180.000} C_DIS
LIN {X 87.767,Y 100.293,Z 78.000,A 180.000,B 0.000,C 180.000} C_DIS
LIN {X 87.779,Y 100.338,Z 78.000,A 180.000,B 0.000,C 180.000} C_DIS
LIN {X 87.821,Y 100.472,Z 78.000,A 180.000,B 0.000,C 180.000} C_DIS
LIN {X 87.878,Y 100.651,Z 78.000,A 180.000,B 0.000,C 180.000} C_DIS
LIN {X 87.936,Y 100.829,Z 78.000,A 180.000,B 0.000,C 180.000} C_DIS
LIN {X 87.958,Y 100.889,Z 78.000,A 180.000,B 0.000,C 180.000} C_DIS
LIN {X 88.072,Y 101.187,Z 78.000,A 180.000,B 0.000,C 180.000} C_DIS
LIN {X 88.137,Y 101.352,Z 78.000,A 180.000,B 0.000,C 180.000} C_DIS
LIN {X 88.142,Y 101.366,Z 78.000,A 180.000,B 0.000,C 180.000} C_DIS
LIN {X 88.218,Y 101.545,Z 78.000,A 180.000,B 0.000,C 180.000} C_DIS
LIN {X 88.316,Y 101.762,Z 78.000,A 180.000,B 0.000,C 180.000} C_DIS
LIN {X 88.380,Y 101.902,Z 78.000,A 180.000,B 0.000,C 180.000} C_DIS
LIN {X 88.472,Y 102.081,Z 78.000,A 180.000,B 0.000,C 180.000} C_DIS
LIN {X 88.564,Y 102.260,Z 78.000,A 180.000,B 0.000,C 180.000} C_DIS
LIN {X 88.661,Y 102.438,Z 78.000,A 180.000,B 0.000,C 180.000} C_DIS
LIN {X 88.673,Y 102.460,Z 78.000,A 180.000,B 0.000,C 180.000} C_DIS
LIN {X 88.765,Y 102.617,Z 78.000,A 180.000,B 0.000,C 180.000} C_DIS
LIN {X 88.870,Y 102.796,Z 78.000,A 180.000,B 0.000,C 180.000} C_DIS
LIN {X 88.982,Y 102.975,Z 78.000,A 180.000,B 0.000,C 180.000} C_DIS
LIN {X 89.101,Y 103.153,Z 78.000,A 180.000,B 0.000,C 180.000} C_DIS
LIN {X 89.209,Y 103.313,Z 78.000,A 180.000,B 0.000,C 180.000} C_DIS
LIN {X 89.223,Y 103.332,Z 78.000,A 180.000,B 0.000,C 180.000} C_DIS
LIN {X 89.354,Y 103.511,Z 78.000,A 180.000,B 0.000,C 180.000} C_DIS
LIN {X 89.489,Y 103.690,Z 78.000,A 180.000,B 0.000,C 180.000} C_DIS
LIN {X 89.567,Y 103.794,Z 78.000,A 180.000,B 0.000,C 180.000} C_DIS
LIN {X 89.627,Y 103.869,Z 78.000,A 180.000,B 0.000,C 180.000} C_DIS
LIN {X 89.746,Y 104.010,Z 78.000,A 180.000,B 0.000,C 180.000} C_DIS
LIN {X 89.777,Y 104.047,Z 78.000,A 180.000,B 0.000,C 180.000} C_DIS
LIN {X 89.925,Y 104.220,Z 78.000,A 180.000,B 0.000,C 180.000} C_DIS
LIN {X 89.930,Y 104.226,Z 78.000,A 180.000,B 0.000,C 180.000} C_DIS
LIN {X 90.098,Y 104.405,Z 78.000,A 180.000,B 0.000,C 180.000} C_DIS
LIN {X 90.282,Y 104.600,Z 78.000,A 180.000,B 0.000,C 180.000} C_DIS
LIN {X 90.444,Y 104.762,Z 78.000,A 180.000,B 0.000,C 180.000} C_DIS
LIN {X 90.640,Y 104.947,Z 78.000,A 180.000,B 0.000,C 180.000} C_DIS
LIN {X 90.818,Y 105.107,Z 78.000,A 180.000,B 0.000,C 180.000} C_DIS
LIN {X 91.045,Y 105.299,Z 78.000,A 180.000,B 0.000,C 180.000} C_DIS
LIN {X 91.176,Y 105.407,Z 78.000,A 180.000,B 0.000,C 180.000} C_DIS
LIN {X 91.263,Y 105.477,Z 78.000,A 180.000,B 0.000,C 180.000} C_DIS
LIN {X 91.355,Y 105.546,Z 78.000,A 180.000,B 0.000,C 180.000} C_DIS
LIN {X 91.533,Y 105.681,Z 78.000,A 180.000,B 0.000,C 180.000} C_DIS
LIN {X 91.712,Y 105.808,Z 78.000,A 180.000,B 0.000,C 180.000} C_DIS
LIN {X 91.891,Y 105.928,Z 78.000,A 180.000,B 0.000,C 180.000} C_DIS
LIN {X 92.020,Y 106.014,Z 78.000,A 180.000,B 0.000,C 180.000} C_DIS
LIN {X 92.070,Y 106.045,Z 78.000,A 180.000,B 0.000,C 180.000} C_DIS
LIN {X 92.249,Y 106.156,Z 78.000,A 180.000,B 0.000,C 180.000} C_DIS
LIN {X 92.427,Y 106.262,Z 78.000,A 180.000,B 0.000,C 180.000} C_DIS
LIN {X 92.606,Y 106.366,Z 78.000,A 180.000,B 0.000,C 180.000} C_DIS
LIN {X 92.616,Y 106.371,Z 78.000,A 180.000,B 0.000,C 180.000} C_DIS
LIN {X 92.785,Y 106.459,Z 78.000,A 180.000,B 0.000,C 180.000} C_DIS
LIN {X 92.964,Y 106.552,Z 78.000,A 180.000,B 0.000,C 180.000} C_DIS
LIN {X 93.142,Y 106.639,Z 78.000,A 180.000,B 0.000,C 180.000} C_DIS
LIN {X 93.321,Y 106.721,Z 78.000,A 180.000,B 0.000,C 180.000} C_DIS
LIN {X 93.500,Y 106.801,Z 78.000,A 180.000,B 0.000,C 180.000} C_DIS
LIN {X 93.679,Y 106.878,Z 78.000,A 180.000,B 0.000,C 180.000} C_DIS
LIN {X 93.756,Y 106.908,Z 78.000,A 180.000,B 0.000,C 180.000} C_DIS
LIN {X 94.036,Y 107.015,Z 78.000,A 180.000,B 0.000,C 180.000} C_DIS
LIN {X 94.170,Y 107.061,Z 78.000,A 180.000,B 0.000,C 180.000} C_DIS
LIN {X 94.215,Y 107.077,Z 78.000,A 180.000,B 0.000,C 180.000} C_DIS
LIN {X 94.245,Y 107.086,Z 78.000,A 180.000,B 0.000,C 180.000} C_DIS
LIN {X 94.394,Y 107.134,Z 78.000,A 180.000,B 0.000,C 180.000} C_DIS
LIN {X 94.573,Y 107.191,Z 78.000,A 180.000,B 0.000,C 180.000} C_DIS
LIN {X 94.751,Y 107.246,Z 78.000,A 180.000,B 0.000,C 180.000} C_DIS
LIN {X 94.822,Y 107.265,Z 78.000,A 180.000,B 0.000,C 180.000} C_DIS
LIN {X 95.109,Y 107.339,Z 78.000,A 180.000,B 0.000,C 180.000} C_DIS
LIN {X 95.288,Y 107.381,Z 78.000,A 180.000,B 0.000,C 180.000} C_DIS
LIN {X 95.604,Y 107.444,Z 78.000,A 180.000,B 0.000,C 180.000} C_DIS
LIN {X 95.645,Y 107.452,Z 78.000,A 180.000,B 0.000,C 180.000} C_DIS
LIN {X 95.824,Y 107.486,Z 78.000,A 180.000,B 0.000,C 180.000} C_DIS
LIN {X 96.003,Y 107.513,Z 78.000,A 180.000,B 0.000,C 180.000} C_DIS
LIN {X 96.181,Y 107.539,Z 78.000,A 180.000,B 0.000,C 180.000} C_DIS
LIN {X 96.360,Y 107.563,Z 78.000,A 180.000,B 0.000,C 180.000} C_DIS
LIN {X 96.539,Y 107.578,Z 78.000,A 180.000,B 0.000,C 180.000} C_DIS
LIN {X 96.718,Y 107.593,Z 78.000,A 180.000,B 0.000,C 180.000} C_DIS
LIN {X 96.897,Y 107.607,Z 78.000,A 180.000,B 0.000,C 180.000} C_DIS
LIN {X 97.075,Y 107.616,Z 78.000,A 180.000,B 0.000,C 180.000} C_DIS
LIN {X 97.433,Y 107.626,Z 78.000,A 180.000,B 0.000,C 180.000} C_DIS
LIN {X 97.612,Y 107.625,Z 78.000,A 180.000,B 0.000,C 180.000} C_DIS
LIN {X 97.790,Y 107.620,Z 78.000,A 180.000,B 0.000,C 180.000} C_DIS
LIN {X 97.969,Y 107.615,Z 78.000,A 180.000,B 0.000,C 180.000} C_DIS
LIN {X 98.148,Y 107.604,Z 78.000,A 180.000,B 0.000,C 180.000} C_DIS
LIN {X 98.327,Y 107.590,Z 78.000,A 180.000,B 0.000,C 180.000} C_DIS
LIN {X 98.505,Y 107.575,Z 78.000,A 180.000,B 0.000,C 180.000} C_DIS
LIN {X 98.684,Y 107.557,Z 78.000,A 180.000,B 0.000,C 180.000} C_DIS
LIN {X 98.863,Y 107.532,Z 78.000,A 180.000,B 0.000,C 180.000} C_DIS
LIN {X 99.042,Y 107.507,Z 78.000,A 180.000,B 0.000,C 180.000} C_DIS
LIN {X 99.221,Y 107.478,Z 78.000,A 180.000,B 0.000,C 180.000} C_DIS
LIN {X 99.396,Y 107.444,Z 78.000,A 180.000,B 0.000,C 180.000} C_DIS
LIN {X 99.578,Y 107.408,Z 78.000,A 180.000,B 0.000,C 180.000} C_DIS
LIN {X 99.757,Y 107.372,Z 78.000,A 180.000,B 0.000,C 180.000} C_DIS
LIN {X 99.936,Y 107.328,Z 78.000,A 180.000,B 0.000,C 180.000} C_DIS
LIN {X 100.178,Y 107.265,Z 78.000,A 180.000,B 0.000,C 180.000} C_DIS
LIN {X 100.293,Y 107.234,Z 78.000,A 180.000,B 0.000,C 180.000} C_DIS
LIN {X 100.472,Y 107.177,Z 78.000,A 180.000,B 0.000,C 180.000} C_DIS
LIN {X 100.651,Y 107.120,Z 78.000,A 180.000,B 0.000,C 180.000} C_DIS
LIN {X 100.755,Y 107.086,Z 78.000,A 180.000,B 0.000,C 180.000} C_DIS
LIN {X 100.829,Y 107.062,Z 78.000,A 180.000,B 0.000,C 180.000} C_DIS
LIN {X 101.008,Y 106.998,Z 78.000,A 180.000,B 0.000,C 180.000} C_DIS
LIN {X 101.244,Y 106.908,Z 78.000,A 180.000,B 0.000,C 180.000} C_DIS
LIN {X 101.366,Y 106.860,Z 78.000,A 180.000,B 0.000,C 180.000} C_DIS
LIN {X 101.545,Y 106.781,Z 78.000,A 180.000,B 0.000,C 180.000} C_DIS
LIN {X 101.723,Y 106.701,Z 78.000,A 180.000,B 0.000,C 180.000} C_DIS
LIN {X 101.902,Y 106.618,Z 78.000,A 180.000,B 0.000,C 180.000} C_DIS
LIN {X 102.040,Y 106.550,Z 78.000,A 180.000,B 0.000,C 180.000} C_DIS
LIN {X 102.260,Y 106.436,Z 78.000,A 180.000,B 0.000,C 180.000} C_DIS
LIN {X 102.384,Y 106.371,Z 78.000,A 180.000,B 0.000,C 180.000} C_DIS
LIN {X 102.438,Y 106.341,Z 78.000,A 180.000,B 0.000,C 180.000} C_DIS
LIN {X 102.617,Y 106.236,Z 78.000,A 180.000,B 0.000,C 180.000} C_DIS
LIN {X 102.690,Y 106.193,Z 78.000,A 180.000,B 0.000,C 180.000} C_DIS
LIN {X 102.796,Y 106.130,Z 78.000,A 180.000,B 0.000,C 180.000} C_DIS
LIN {X 102.975,Y 106.017,Z 78.000,A 180.000,B 0.000,C 180.000} C_DIS
LIN {X 102.980,Y 106.014,Z 78.000,A 180.000,B 0.000,C 180.000} C_DIS
LIN {X 103.153,Y 105.898,Z 78.000,A 180.000,B 0.000,C 180.000} C_DIS
LIN {X 103.248,Y 105.835,Z 78.000,A 180.000,B 0.000,C 180.000} C_DIS
LIN {X 103.332,Y 105.778,Z 78.000,A 180.000,B 0.000,C 180.000} C_DIS
LIN {X 103.499,Y 105.656,Z 78.000,A 180.000,B 0.000,C 180.000} C_DIS
LIN {X 103.690,Y 105.513,Z 78.000,A 180.000,B 0.000,C 180.000} C_DIS
LIN {X 103.737,Y 105.477,Z 78.000,A 180.000,B 0.000,C 180.000} C_DIS
LIN {X 103.869,Y 105.370,Z 78.000,A 180.000,B 0.000,C 180.000} C_DIS
LIN {X 103.955,Y 105.299,Z 78.000,A 180.000,B 0.000,C 180.000} C_DIS
LIN {X 104.166,Y 105.120,Z 78.000,A 180.000,B 0.000,C 180.000} C_DIS
LIN {X 104.226,Y 105.069,Z 78.000,A 180.000,B 0.000,C 180.000} C_DIS
LIN {X 104.367,Y 104.941,Z 78.000,A 180.000,B 0.000,C 180.000} C_DIS
LIN {X 104.584,Y 104.736,Z 78.000,A 180.000,B 0.000,C 180.000} C_DIS
LIN {X 104.733,Y 104.584,Z 78.000,A 180.000,B 0.000,C 180.000} C_DIS
LIN {X 104.902,Y 104.405,Z 78.000,A 180.000,B 0.000,C 180.000} C_DIS
LIN {X 104.941,Y 104.363,Z 78.000,A 180.000,B 0.000,C 180.000} C_DIS
LIN {X 105.070,Y 104.226,Z 78.000,A 180.000,B 0.000,C 180.000} C_DIS
LIN {X 105.120,Y 104.169,Z 78.000,A 180.000,B 0.000,C 180.000} C_DIS
LIN {X 105.223,Y 104.047,Z 78.000,A 180.000,B 0.000,C 180.000} C_DIS
LIN {X 105.299,Y 103.957,Z 78.000,A 180.000,B 0.000,C 180.000} C_DIS
LIN {X 105.373,Y 103.869,Z 78.000,A 180.000,B 0.000,C 180.000} C_DIS
LIN {X 105.477,Y 103.735,Z 78.000,A 180.000,B 0.000,C 180.000} C_DIS
LIN {X 105.656,Y 103.497,Z 78.000,A 180.000,B 0.000,C 180.000} C_DIS
LIN {X 105.777,Y 103.332,Z 78.000,A 180.000,B 0.000,C 180.000} C_DIS
LIN {X 105.835,Y 103.249,Z 78.000,A 180.000,B 0.000,C 180.000} C_DIS
LIN {X 106.018,Y 102.975,Z 78.000,A 180.000,B 0.000,C 180.000} C_DIS
LIN {X 106.130,Y 102.796,Z 78.000,A 180.000,B 0.000,C 180.000} C_DIS
LIN {X 106.235,Y 102.617,Z 78.000,A 180.000,B 0.000,C 180.000} C_DIS
LIN {X 106.339,Y 102.438,Z 78.000,A 180.000,B 0.000,C 180.000} C_DIS
LIN {X 106.371,Y 102.379,Z 78.000,A 180.000,B 0.000,C 180.000} C_DIS
LIN {X 106.436,Y 102.260,Z 78.000,A 180.000,B 0.000,C 180.000} C_DIS
LIN {X 106.550,Y 102.039,Z 78.000,A 180.000,B 0.000,C 180.000} C_DIS
LIN {X 106.620,Y 101.902,Z 78.000,A 180.000,B 0.000,C 180.000} C_DIS
LIN {X 106.702,Y 101.723,Z 78.000,A 180.000,B 0.000,C 180.000} C_DIS
LIN {X 106.782,Y 101.545,Z 78.000,A 180.000,B 0.000,C 180.000} C_DIS
LIN {X 106.858,Y 101.366,Z 78.000,A 180.000,B 0.000,C 180.000} C_DIS
LIN {X 106.908,Y 101.240,Z 78.000,A 180.000,B 0.000,C 180.000} C_DIS
LIN {X 106.928,Y 101.187,Z 78.000,A 180.000,B 0.000,C 180.000} C_DIS
LIN {X 106.996,Y 101.008,Z 78.000,A 180.000,B 0.000,C 180.000} C_DIS
LIN {X 107.064,Y 100.829,Z 78.000,A 180.000,B 0.000,C 180.000} C_DIS
LIN {X 107.086,Y 100.763,Z 78.000,A 180.000,B 0.000,C 180.000} C_DIS
LIN {X 107.122,Y 100.651,Z 78.000,A 180.000,B 0.000,C 180.000} C_DIS
LIN {X 107.179,Y 100.472,Z 78.000,A 180.000,B 0.000,C 180.000} C_DIS
LIN {X 107.233,Y 100.293,Z 78.000,A 180.000,B 0.000,C 180.000} C_DIS
LIN {X 107.265,Y 100.169,Z 78.000,A 180.000,B 0.000,C 180.000} C_DIS
LIN {X 107.325,Y 99.936,Z 78.000,A 180.000,B 0.000,C 180.000} C_DIS
LIN {X 107.371,Y 99.757,Z 78.000,A 180.000,B 0.000,C 180.000} C_DIS
LIN {X 107.409,Y 99.578,Z 78.000,A 180.000,B 0.000,C 180.000} C_DIS
LIN {X 107.445,Y 99.399,Z 78.000,A 180.000,B 0.000,C 180.000} C_DIS
LIN {X 107.480,Y 99.221,Z 78.000,A 180.000,B 0.000,C 180.000} C_DIS
LIN {X 107.506,Y 99.042,Z 78.000,A 180.000,B 0.000,C 180.000} C_DIS
LIN {X 107.531,Y 98.863,Z 78.000,A 180.000,B 0.000,C 180.000} C_DIS
LIN {X 107.555,Y 98.684,Z 78.000,A 180.000,B 0.000,C 180.000} C_DIS
LIN {X 107.575,Y 98.505,Z 78.000,A 180.000,B 0.000,C 180.000} C_DIS
LIN {X 107.606,Y 98.148,Z 78.000,A 180.000,B 0.000,C 180.000} C_DIS
LIN {X 107.615,Y 97.969,Z 78.000,A 180.000,B 0.000,C 180.000} C_DIS
LIN {X 107.623,Y 97.680,Z 78.000,A 180.000,B 0.000,C 180.000} C_DIS
LIN {X 107.624,Y 97.612,Z 78.000,A 180.000,B 0.000,C 180.000} C_DIS
LIN {X 107.625,Y 97.433,Z 78.000,A 180.000,B 0.000,C 180.000} C_DIS
LIN {X 107.623,Y 97.320,Z 78.000,A 180.000,B 0.000,C 180.000} C_DIS
LIN {X 107.616,Y 97.075,Z 78.000,A 180.000,B 0.000,C 180.000} C_DIS
LIN {X 107.609,Y 96.897,Z 78.000,A 180.000,B 0.000,C 180.000} C_DIS
LIN {X 107.594,Y 96.718,Z 78.000,A 180.000,B 0.000,C 180.000} C_DIS
LIN {X 107.579,Y 96.539,Z 78.000,A 180.000,B 0.000,C 180.000} C_DIS
LIN {X 107.561,Y 96.360,Z 78.000,A 180.000,B 0.000,C 180.000} C_DIS
LIN {X 107.537,Y 96.181,Z 78.000,A 180.000,B 0.000,C 180.000} C_DIS
LIN {X 107.512,Y 96.003,Z 78.000,A 180.000,B 0.000,C 180.000} C_DIS
LIN {X 107.487,Y 95.824,Z 78.000,A 180.000,B 0.000,C 180.000} C_DIS
LIN {X 107.454,Y 95.645,Z 78.000,A 180.000,B 0.000,C 180.000} C_DIS
LIN {X 107.418,Y 95.466,Z 78.000,A 180.000,B 0.000,C 180.000} C_DIS
LIN {X 107.382,Y 95.288,Z 78.000,A 180.000,B 0.000,C 180.000} C_DIS
LIN {X 107.337,Y 95.109,Z 78.000,A 180.000,B 0.000,C 180.000} C_DIS
LIN {X 107.291,Y 94.930,Z 78.000,A 180.000,B 0.000,C 180.000} C_DIS
LIN {X 107.245,Y 94.751,Z 78.000,A 180.000,B 0.000,C 180.000} C_DIS
LIN {X 107.193,Y 94.573,Z 78.000,A 180.000,B 0.000,C 180.000} C_DIS
LIN {X 107.136,Y 94.394,Z 78.000,A 180.000,B 0.000,C 180.000} C_DIS
LIN {X 107.086,Y 94.237,Z 78.000,A 180.000,B 0.000,C 180.000} C_DIS
LIN {X 107.079,Y 94.215,Z 78.000,A 180.000,B 0.000,C 180.000} C_DIS
LIN {X 107.013,Y 94.036,Z 78.000,A 180.000,B 0.000,C 180.000} C_DIS
LIN {X 106.945,Y 93.857,Z 78.000,A 180.000,B 0.000,C 180.000} C_DIS
LIN {X 106.908,Y 93.760,Z 78.000,A 180.000,B 0.000,C 180.000} C_DIS
LIN {X 106.876,Y 93.679,Z 78.000,A 180.000,B 0.000,C 180.000} C_DIS
LIN {X 106.802,Y 93.500,Z 78.000,A 180.000,B 0.000,C 180.000} C_DIS
LIN {X 106.722,Y 93.321,Z 78.000,A 180.000,B 0.000,C 180.000} C_DIS
LIN {X 106.641,Y 93.142,Z 78.000,A 180.000,B 0.000,C 180.000} C_DIS
LIN {X 106.551,Y 92.964,Z 78.000,A 180.000,B 0.000,C 180.000} C_DIS
LIN {X 106.459,Y 92.785,Z 78.000,A 180.000,B 0.000,C 180.000} C_DIS
LIN {X 106.371,Y 92.621,Z 78.000,A 180.000,B 0.000,C 180.000} C_DIS
LIN {X 106.363,Y 92.606,Z 78.000,A 180.000,B 0.000,C 180.000} C_DIS
LIN {X 106.262,Y 92.427,Z 78.000,A 180.000,B 0.000,C 180.000} C_DIS
LIN {X 106.156,Y 92.249,Z 78.000,A 180.000,B 0.000,C 180.000} C_DIS
LIN {X 106.048,Y 92.070,Z 78.000,A 180.000,B 0.000,C 180.000} C_DIS
LIN {X 106.014,Y 92.019,Z 78.000,A 180.000,B 0.000,C 180.000} C_DIS
LIN {X 105.835,Y 91.751,Z 78.000,A 180.000,B 0.000,C 180.000} C_DIS
LIN {X 105.808,Y 91.712,Z 78.000,A 180.000,B 0.000,C 180.000} C_DIS
LIN {X 105.679,Y 91.533,Z 78.000,A 180.000,B 0.000,C 180.000} C_DIS
LIN {X 105.656,Y 91.503,Z 78.000,A 180.000,B 0.000,C 180.000} C_DIS
LIN {X 105.477,Y 91.265,Z 78.000,A 180.000,B 0.000,C 180.000} C_DIS
LIN {X 105.409,Y 91.176,Z 78.000,A 180.000,B 0.000,C 180.000} C_DIS
LIN {X 105.299,Y 91.043,Z 78.000,A 180.000,B 0.000,C 180.000} C_DIS
LIN {X 105.260,Y 90.997,Z 78.000,A 180.000,B 0.000,C 180.000} C_DIS
LIN {X 105.120,Y 90.831,Z 78.000,A 180.000,B 0.000,C 180.000} C_DIS
LIN {X 105.109,Y 90.818,Z 78.000,A 180.000,B 0.000,C 180.000} C_DIS
LIN {X 104.944,Y 90.640,Z 78.000,A 180.000,B 0.000,C 180.000} C_DIS
LIN {X 104.941,Y 90.637,Z 78.000,A 180.000,B 0.000,C 180.000} C_DIS
LIN {X 104.762,Y 90.447,Z 78.000,A 180.000,B 0.000,C 180.000} C_DIS
LIN {X 104.602,Y 90.282,Z 78.000,A 180.000,B 0.000,C 180.000} C_DIS
LIN {X 104.584,Y 90.264,Z 78.000,A 180.000,B 0.000,C 180.000} C_DIS
LIN {X 104.405,Y 90.095,Z 78.000,A 180.000,B 0.000,C 180.000} C_DIS
LIN {X 104.226,Y 89.931,Z 78.000,A 180.000,B 0.000,C 180.000} C_DIS
LIN {X 104.219,Y 89.925,Z 78.000,A 180.000,B 0.000,C 180.000} C_DIS
LIN {X 104.007,Y 89.746,Z 78.000,A 180.000,B 0.000,C 180.000} C_DIS
LIN {X 103.869,Y 89.630,Z 78.000,A 180.000,B 0.000,C 180.000} C_DIS
LIN {X 103.793,Y 89.567,Z 78.000,A 180.000,B 0.000,C 180.000} C_DIS
LIN {X 103.690,Y 89.487,Z 78.000,A 180.000,B 0.000,C 180.000} C_DIS
LIN {X 103.511,Y 89.353,Z 78.000,A 180.000,B 0.000,C 180.000} C_DIS
LIN {X 103.332,Y 89.222,Z 78.000,A 180.000,B 0.000,C 180.000} C_DIS
LIN {X 103.314,Y 89.209,Z 78.000,A 180.000,B 0.000,C 180.000} C_DIS
LIN {X 103.047,Y 89.031,Z 78.000,A 180.000,B 0.000,C 180.000} C_DIS
LIN {X 102.975,Y 88.983,Z 78.000,A 180.000,B 0.000,C 180.000} C_DIS
LIN {X 102.796,Y 88.870,Z 78.000,A 180.000,B 0.000,C 180.000} C_DIS
LIN {X 102.765,Y 88.852,Z 78.000,A 180.000,B 0.000,C 180.000} C_DIS
LIN {X 102.462,Y 88.673,Z 78.000,A 180.000,B 0.000,C 180.000} C_DIS
LIN {X 102.438,Y 88.659,Z 78.000,A 180.000,B 0.000,C 180.000} C_DIS
LIN {X 102.260,Y 88.564,Z 78.000,A 180.000,B 0.000,C 180.000} C_DIS
LIN {X 102.081,Y 88.471,Z 78.000,A 180.000,B 0.000,C 180.000} C_DIS
LIN {X 101.902,Y 88.382,Z 78.000,A 180.000,B 0.000,C 180.000} C_DIS
LIN {X 101.760,Y 88.316,Z 78.000,A 180.000,B 0.000,C 180.000} C_DIS
LIN {X 101.723,Y 88.299,Z 78.000,A 180.000,B 0.000,C 180.000} C_DIS
LIN {X 101.545,Y 88.219,Z 78.000,A 180.000,B 0.000,C 180.000} C_DIS
LIN {X 101.366,Y 88.140,Z 78.000,A 180.000,B 0.000,C 180.000} C_DIS
LIN {X 101.358,Y 88.137,Z 78.000,A 180.000,B 0.000,C 180.000} C_DIS
LIN {X 101.187,Y 88.070,Z 78.000,A 180.000,B 0.000,C 180.000} C_DIS
LIN {X 101.008,Y 88.002,Z 78.000,A 180.000,B 0.000,C 180.000} C_DIS
LIN {X 100.890,Y 87.958,Z 78.000,A 180.000,B 0.000,C 180.000} C_DIS
LIN {X 100.829,Y 87.938,Z 78.000,A 180.000,B 0.000,C 180.000} C_DIS
LIN {X 100.651,Y 87.880,Z 78.000,A 180.000,B 0.000,C 180.000} C_DIS
LIN {X 100.335,Y 87.779,Z 78.000,A 180.000,B 0.000,C 180.000} C_DIS
LIN {X 100.293,Y 87.766,Z 78.000,A 180.000,B 0.000,C 180.000} C_DIS
LIN {X 100.114,Y 87.718,Z 78.000,A 180.000,B 0.000,C 180.000} C_DIS
LIN {X 99.936,Y 87.672,Z 78.000,A 180.000,B 0.000,C 180.000} C_DIS
LIN {X 99.757,Y 87.628,Z 78.000,A 180.000,B 0.000,C 180.000} C_DIS
LIN {X 99.619,Y 87.601,Z 78.000,A 180.000,B 0.000,C 180.000} C_DIS
LIN {X 99.399,Y 87.557,Z 78.000,A 180.000,B 0.000,C 180.000} C_DIS
LIN {X 99.221,Y 87.522,Z 78.000,A 180.000,B 0.000,C 180.000} C_DIS
LIN {X 99.042,Y 87.493,Z 78.000,A 180.000,B 0.000,C 180.000} C_DIS
LIN {X 98.863,Y 87.468,Z 78.000,A 180.000,B 0.000,C 180.000} C_DIS
LIN {X 98.684,Y 87.443,Z 78.000,A 180.000,B 0.000,C 180.000} C_DIS
LIN {X 98.505,Y 87.425,Z 78.000,A 180.000,B 0.000,C 180.000} C_DIS
LIN {X 98.327,Y 87.410,Z 78.000,A 180.000,B 0.000,C 180.000} C_DIS
LIN {X 98.148,Y 87.396,Z 78.000,A 180.000,B 0.000,C 180.000} C_DIS
LIN {X 97.969,Y 87.385,Z 78.000,A 180.000,B 0.000,C 180.000} C_DIS
LIN {X 97.790,Y 87.380,Z 78.000,A 180.000,B 0.000,C 180.000} C_DIS
LIN {X 97.612,Y 87.375,Z 78.000,A 180.000,B 0.000,C 180.000} C_DIS
LIN {X 97.433,Y 87.374,Z 78.000,A 180.000,B 0.000,C 180.000} C_DIS
LIN {X 97.075,Y 87.384,Z 78.000,A 180.000,B 0.000,C 180.000} C_DIS
LIN {X 96.897,Y 87.393,Z 78.000,A 180.000,B 0.000,C 180.000} C_DIS
LIN {X 96.718,Y 87.407,Z 78.000,A 180.000,B 0.000,C 180.000} C_DIS
LIN {X 96.538,Y 87.422,Z 78.000,A 180.000,B 0.000,C 180.000} C_DIS
LIN {X 96.360,Y 87.437,Z 78.000,A 180.000,B 0.000,C 180.000} C_DIS
LIN {X 96.181,Y 87.461,Z 78.000,A 180.000,B 0.000,C 180.000} C_DIS
LIN {X 96.003,Y 87.487,Z 78.000,A 180.000,B 0.000,C 180.000} C_DIS
LIN {X 95.824,Y 87.514,Z 78.000,A 180.000,B 0.000,C 180.000} C_DIS
LIN {X 95.645,Y 87.548,Z 78.000,A 180.000,B 0.000,C 180.000} C_DIS
LIN {X 95.466,Y 87.584,Z 78.000,A 180.000,B 0.000,C 180.000} C_DIS
LIN {X 95.288,Y 87.619,Z 78.000,A 180.000,B 0.000,C 180.000} C_DIS
LIN {X 95.109,Y 87.661,Z 78.000,A 180.000,B 0.000,C 180.000} C_DIS
LIN {X 94.930,Y 87.707,Z 78.000,A 180.000,B 0.000,C 180.000} C_DIS
LIN {X 94.776,Y 87.747,Z 78.000,A 180.000,B 0.000,C 180.000} C_DIS
; Link Move Starts
LIN {X 94.494,Y 87.831,Z 78.000,A 180.000,B 0.000,C 180.000} C_DIS
LIN {X 94.196,Y 87.927,Z 77.999,A 180.000,B 0.000,C 180.000} C_DIS
LIN {X 93.923,Y 88.025,Z 77.998,A 180.000,B 0.000,C 180.000} C_DIS
LIN {X 93.647,Y 88.130,Z 77.997,A 180.000,B 0.000,C 180.000} C_DIS
LIN {X 93.364,Y 88.255,Z 77.995,A 180.000,B 0.000,C 180.000} C_DIS
LIN {X 93.092,Y 88.378,Z 77.992,A 180.000,B 0.000,C 180.000} C_DIS
LIN {X 92.819,Y 88.515,Z 77.989,A 180.000,B 0.000,C 180.000} C_DIS
LIN {X 92.557,Y 88.652,Z 77.986,A 180.000,B 0.000,C 180.000} C_DIS
LIN {X 92.293,Y 88.806,Z 77.983,A 180.000,B 0.000,C 180.000} C_DIS
LIN {X 92.037,Y 88.961,Z 77.979,A 180.000,B 0.000,C 180.000} C_DIS
LIN {X 91.781,Y 89.129,Z 77.974,A 180.000,B 0.000,C 180.000} C_DIS
LIN {X 91.539,Y 89.294,Z 77.970,A 180.000,B 0.000,C 180.000} C_DIS
LIN {X 91.414,Y 89.387,Z 77.967,A 180.000,B 0.000,C 180.000} C_DIS
LIN {X 91.288,Y 89.481,Z 77.964,A 180.000,B 0.000,C 180.000} C_DIS
LIN {X 91.173,Y 89.570,Z 77.962,A 180.000,B 0.000,C 180.000} C_DIS
LIN {X 91.060,Y 89.661,Z 77.959,A 180.000,B 0.000,C 180.000} C_DIS
LIN {X 90.939,Y 89.762,Z 77.956,A 180.000,B 0.000,C 180.000} C_DIS
LIN {X 90.818,Y 89.862,Z 77.953,A 180.000,B 0.000,C 180.000} C_DIS
LIN {X 90.705,Y 89.957,Z 77.950,A 180.000,B 0.000,C 180.000} C_DIS
LIN {X 90.596,Y 90.057,Z 77.947,A 180.000,B 0.000,C 180.000} C_DIS
LIN {X 90.488,Y 90.157,Z 77.944,A 180.000,B 0.000,C 180.000} C_DIS
LIN {X 90.381,Y 90.257,Z 77.941,A 180.000,B 0.000,C 180.000} C_DIS
LIN {X 90.272,Y 90.365,Z 77.937,A 180.000,B 0.000,C 180.000} C_DIS
LIN {X 90.166,Y 90.475,Z 77.934,A 180.000,B 0.000,C 180.000} C_DIS
LIN {X 90.057,Y 90.588,Z 77.930,A 180.000,B 0.000,C 180.000} C_DIS
LIN {X 89.949,Y 90.700,Z 77.927,A 180.000,B 0.000,C 180.000} C_DIS
LIN {X 89.850,Y 90.808,Z 77.923,A 180.000,B 0.000,C 180.000} C_DIS
LIN {X 89.754,Y 90.919,Z 77.919,A 180.000,B 0.000,C 180.000} C_DIS
LIN {X 89.653,Y 91.035,Z 77.916,A 180.000,B 0.000,C 180.000} C_DIS
LIN {X 89.554,Y 91.152,Z 77.912,A 180.000,B 0.000,C 180.000} C_DIS
LIN {X 89.462,Y 91.270,Z 77.908,A 180.000,B 0.000,C 180.000} C_DIS
LIN {X 89.371,Y 91.388,Z 77.904,A 180.000,B 0.000,C 180.000} C_DIS
LIN {X 89.280,Y 91.506,Z 77.900,A 180.000,B 0.000,C 180.000} C_DIS
LIN {X 89.191,Y 91.625,Z 77.896,A 180.000,B 0.000,C 180.000} C_DIS
LIN {X 89.101,Y 91.751,Z 77.891,A 180.000,B 0.000,C 180.000} C_DIS
LIN {X 89.014,Y 91.879,Z 77.887,A 180.000,B 0.000,C 180.000} C_DIS
LIN {X 88.930,Y 92.000,Z 77.883,A 180.000,B 0.000,C 180.000} C_DIS
LIN {X 88.849,Y 92.123,Z 77.878,A 180.000,B 0.000,C 180.000} C_DIS
LIN {X 88.768,Y 92.256,Z 77.874,A 180.000,B 0.000,C 180.000} C_DIS
LIN {X 88.687,Y 92.390,Z 77.869,A 180.000,B 0.000,C 180.000} C_DIS
LIN {X 88.611,Y 92.517,Z 77.864,A 180.000,B 0.000,C 180.000} C_DIS
LIN {X 88.537,Y 92.646,Z 77.860,A 180.000,B 0.000,C 180.000} C_DIS
LIN {X 88.463,Y 92.783,Z 77.855,A 180.000,B 0.000,C 180.000} C_DIS
LIN {X 88.390,Y 92.920,Z 77.850,A 180.000,B 0.000,C 180.000} C_DIS
LIN {X 88.321,Y 93.049,Z 77.845,A 180.000,B 0.000,C 180.000} C_DIS
LIN {X 88.257,Y 93.181,Z 77.840,A 180.000,B 0.000,C 180.000} C_DIS
LIN {X 88.224,Y 93.252,Z 77.838,A 180.000,B 0.000,C 180.000} C_DIS
LIN {X 88.190,Y 93.324,Z 77.835,A 180.000,B 0.000,C 180.000} C_DIS
LIN {X 88.157,Y 93.395,Z 77.832,A 180.000,B 0.000,C 180.000} C_DIS
LIN {X 88.124,Y 93.466,Z 77.830,A 180.000,B 0.000,C 180.000} C_DIS
LIN {X 88.093,Y 93.534,Z 77.827,A 180.000,B 0.000,C 180.000} C_DIS
LIN {X 88.065,Y 93.602,Z 77.825,A 180.000,B 0.000,C 180.000} C_DIS
LIN {X 88.036,Y 93.670,Z 77.822,A 180.000,B 0.000,C 180.000} C_DIS
LIN {X 88.008,Y 93.738,Z 77.820,A 180.000,B 0.000,C 180.000} C_DIS
LIN {X 87.950,Y 93.882,Z 77.814,A 180.000,B 0.000,C 180.000} C_DIS
LIN {X 87.893,Y 94.026,Z 77.809,A 180.000,B 0.000,C 180.000} C_DIS
LIN {X 87.865,Y 94.095,Z 77.806,A 180.000,B 0.000,C 180.000} C_DIS
LIN {X 87.839,Y 94.165,Z 77.804,A 180.000,B 0.000,C 180.000} C_DIS
LIN {X 87.814,Y 94.236,Z 77.801,A 180.000,B 0.000,C 180.000} C_DIS
LIN {X 87.791,Y 94.306,Z 77.799,A 180.000,B 0.000,C 180.000} C_DIS
LIN {X 87.741,Y 94.452,Z 77.793,A 180.000,B 0.000,C 180.000} C_DIS
LIN {X 87.717,Y 94.526,Z 77.791,A 180.000,B 0.000,C 180.000} C_DIS
LIN {X 87.692,Y 94.599,Z 77.788,A 180.000,B 0.000,C 180.000} C_DIS
LIN {X 87.671,Y 94.670,Z 77.785,A 180.000,B 0.000,C 180.000} C_DIS
LIN {X 87.651,Y 94.743,Z 77.783,A 180.000,B 0.000,C 180.000} C_DIS
LIN {X 87.590,Y 94.963,Z 77.775,A 180.000,B 0.000,C 180.000} C_DIS
LIN {X 87.569,Y 95.039,Z 77.772,A 180.000,B 0.000,C 180.000} C_DIS
LIN {X 87.548,Y 95.115,Z 77.769,A 180.000,B 0.000,C 180.000} C_DIS
LIN {X 87.527,Y 95.190,Z 77.766,A 180.000,B 0.000,C 180.000} C_DIS
LIN {X 87.509,Y 95.262,Z 77.764,A 180.000,B 0.000,C 180.000} C_DIS
LIN {X 87.492,Y 95.334,Z 77.761,A 180.000,B 0.000,C 180.000} C_DIS
LIN {X 87.445,Y 95.552,Z 77.753,A 180.000,B 0.000,C 180.000} C_DIS
LIN {X 87.413,Y 95.698,Z 77.748,A 180.000,B 0.000,C 180.000} C_DIS
LIN {X 87.399,Y 95.772,Z 77.746,A 180.000,B 0.000,C 180.000} C_DIS
LIN {X 87.386,Y 95.849,Z 77.743,A 180.000,B 0.000,C 180.000} C_DIS
LIN {X 87.362,Y 96.002,Z 77.737,A 180.000,B 0.000,C 180.000} C_DIS
LIN {X 87.350,Y 96.078,Z 77.735,A 180.000,B 0.000,C 180.000} C_DIS
LIN {X 87.338,Y 96.155,Z 77.732,A 180.000,B 0.000,C 180.000} C_DIS
LIN {X 87.326,Y 96.231,Z 77.729,A 180.000,B 0.000,C 180.000} C_DIS
LIN {X 87.304,Y 96.385,Z 77.724,A 180.000,B 0.000,C 180.000} C_DIS
LIN {X 87.295,Y 96.460,Z 77.721,A 180.000,B 0.000,C 180.000} C_DIS
LIN {X 87.287,Y 96.535,Z 77.719,A 180.000,B 0.000,C 180.000} C_DIS
LIN {X 87.257,Y 96.833,Z 77.708,A 180.000,B 0.000,C 180.000} C_DIS
LIN {X 87.250,Y 96.907,Z 77.706,A 180.000,B 0.000,C 180.000} C_DIS
LIN {X 87.246,Y 96.982,Z 77.703,A 180.000,B 0.000,C 180.000} C_DIS
LIN {X 87.239,Y 97.137,Z 77.698,A 180.000,B 0.000,C 180.000} C_DIS
LIN {X 87.232,Y 97.293,Z 77.692,A 180.000,B 0.000,C 180.000} C_DIS
LIN {X 87.229,Y 97.369,Z 77.689,A 180.000,B 0.000,C 180.000} C_DIS
LIN {X 87.227,Y 97.446,Z 77.687,A 180.000,B 0.000,C 180.000} C_DIS
LIN {X 87.226,Y 97.523,Z 77.684,A 180.000,B 0.000,C 180.000} C_DIS
LIN {X 87.225,Y 97.600,Z 77.681,A 180.000,B 0.000,C 180.000} C_DIS
LIN {X 87.225,Y 97.676,Z 77.679,A 180.000,B 0.000,C 180.000} C_DIS
LIN {X 87.227,Y 97.830,Z 77.673,A 180.000,B 0.000,C 180.000} C_DIS
LIN {X 87.228,Y 97.907,Z 77.671,A 180.000,B 0.000,C 180.000} C_DIS
LIN {X 87.229,Y 97.981,Z 77.668,A 180.000,B 0.000,C 180.000} C_DIS
LIN {X 87.230,Y 98.055,Z 77.665,A 180.000,B 0.000,C 180.000} C_DIS
LIN {X 87.233,Y 98.130,Z 77.663,A 180.000,B 0.000,C 180.000} C_DIS
LIN {X 87.238,Y 98.204,Z 77.660,A 180.000,B 0.000,C 180.000} C_DIS
LIN {X 87.254,Y 98.436,Z 77.652,A 180.000,B 0.000,C 180.000} C_DIS
LIN {X 87.259,Y 98.513,Z 77.649,A 180.000,B 0.000,C 180.000} C_DIS
LIN {X 87.265,Y 98.590,Z 77.647,A 180.000,B 0.000,C 180.000} C_DIS
LIN {X 87.273,Y 98.666,Z 77.644,A 180.000,B 0.000,C 180.000} C_DIS
LIN {X 87.281,Y 98.742,Z 77.641,A 180.000,B 0.000,C 180.000} C_DIS
LIN {X 87.290,Y 98.818,Z 77.639,A 180.000,B 0.000,C 180.000} C_DIS
LIN {X 87.319,Y 99.050,Z 77.631,A 180.000,B 0.000,C 180.000} C_DIS
LIN {X 87.329,Y 99.128,Z 77.628,A 180.000,B 0.000,C 180.000} C_DIS
LIN {X 87.338,Y 99.202,Z 77.625,A 180.000,B 0.000,C 180.000} C_DIS
LIN {X 87.349,Y 99.275,Z 77.623,A 180.000,B 0.000,C 180.000} C_DIS
LIN {X 87.362,Y 99.349,Z 77.620,A 180.000,B 0.000,C 180.000} C_DIS
LIN {X 87.389,Y 99.497,Z 77.615,A 180.000,B 0.000,C 180.000} C_DIS
LIN {X 87.416,Y 99.647,Z 77.609,A 180.000,B 0.000,C 180.000} C_DIS
LIN {X 87.430,Y 99.722,Z 77.607,A 180.000,B 0.000,C 180.000} C_DIS
LIN {X 87.446,Y 99.798,Z 77.604,A 180.000,B 0.000,C 180.000} C_DIS
LIN {X 87.464,Y 99.873,Z 77.601,A 180.000,B 0.000,C 180.000} C_DIS
LIN {X 87.482,Y 99.949,Z 77.599,A 180.000,B 0.000,C 180.000} C_DIS
LIN {X 87.501,Y 100.024,Z 77.596,A 180.000,B 0.000,C 180.000} C_DIS
LIN {X 87.555,Y 100.252,Z 77.588,A 180.000,B 0.000,C 180.000} C_DIS
LIN {X 87.574,Y 100.328,Z 77.585,A 180.000,B 0.000,C 180.000} C_DIS
LIN {X 87.593,Y 100.401,Z 77.582,A 180.000,B 0.000,C 180.000} C_DIS
LIN {X 87.613,Y 100.474,Z 77.580,A 180.000,B 0.000,C 180.000} C_DIS
LIN {X 87.702,Y 100.767,Z 77.569,A 180.000,B 0.000,C 180.000} C_DIS
LIN {X 87.724,Y 100.842,Z 77.566,A 180.000,B 0.000,C 180.000} C_DIS
LIN {X 87.749,Y 100.916,Z 77.564,A 180.000,B 0.000,C 180.000} C_DIS
LIN {X 87.774,Y 100.988,Z 77.561,A 180.000,B 0.000,C 180.000} C_DIS
LIN {X 87.878,Y 101.273,Z 77.550,A 180.000,B 0.000,C 180.000} C_DIS
LIN {X 87.904,Y 101.345,Z 77.548,A 180.000,B 0.000,C 180.000} C_DIS
LIN {X 87.931,Y 101.416,Z 77.545,A 180.000,B 0.000,C 180.000} C_DIS
LIN {X 87.958,Y 101.488,Z 77.542,A 180.000,B 0.000,C 180.000} C_DIS
LIN {X 87.987,Y 101.560,Z 77.540,A 180.000,B 0.000,C 180.000} C_DIS
LIN {X 88.018,Y 101.631,Z 77.537,A 180.000,B 0.000,C 180.000} C_DIS
LIN {X 88.138,Y 101.913,Z 77.526,A 180.000,B 0.000,C 180.000} C_DIS
LIN {X 88.169,Y 101.982,Z 77.524,A 180.000,B 0.000,C 180.000} C_DIS
LIN {X 88.202,Y 102.050,Z 77.521,A 180.000,B 0.000,C 180.000} C_DIS
LIN {X 88.341,Y 102.331,Z 77.510,A 180.000,B 0.000,C 180.000} C_DIS
LIN {X 88.375,Y 102.400,Z 77.507,A 180.000,B 0.000,C 180.000} C_DIS
LIN {X 88.411,Y 102.468,Z 77.505,A 180.000,B 0.000,C 180.000} C_DIS
LIN {X 88.447,Y 102.535,Z 77.502,A 180.000,B 0.000,C 180.000} C_DIS
LIN {X 88.483,Y 102.603,Z 77.499,A 180.000,B 0.000,C 180.000} C_DIS
LIN {X 88.521,Y 102.671,Z 77.497,A 180.000,B 0.000,C 180.000} C_DIS
LIN {X 88.673,Y 102.939,Z 77.486,A 180.000,B 0.000,C 180.000} C_DIS
LIN {X 88.711,Y 103.005,Z 77.483,A 180.000,B 0.000,C 180.000} C_DIS
LIN {X 88.751,Y 103.069,Z 77.480,A 180.000,B 0.000,C 180.000} C_DIS
LIN {X 88.792,Y 103.133,Z 77.478,A 180.000,B 0.000,C 180.000} C_DIS
LIN {X 88.960,Y 103.394,Z 77.467,A 180.000,B 0.000,C 180.000} C_DIS
LIN {X 89.003,Y 103.458,Z 77.464,A 180.000,B 0.000,C 180.000} C_DIS
LIN {X 89.047,Y 103.521,Z 77.462,A 180.000,B 0.000,C 180.000} C_DIS
LIN {X 89.091,Y 103.584,Z 77.459,A 180.000,B 0.000,C 180.000} C_DIS
LIN {X 89.136,Y 103.647,Z 77.456,A 180.000,B 0.000,C 180.000} C_DIS
LIN {X 89.321,Y 103.901,Z 77.445,A 180.000,B 0.000,C 180.000} C_DIS
LIN {X 89.366,Y 103.962,Z 77.443,A 180.000,B 0.000,C 180.000} C_DIS
LIN {X 89.412,Y 104.022,Z 77.440,A 180.000,B 0.000,C 180.000} C_DIS
LIN {X 89.460,Y 104.081,Z 77.437,A 180.000,B 0.000,C 180.000} C_DIS
LIN {X 89.657,Y 104.322,Z 77.426,A 180.000,B 0.000,C 180.000} C_DIS
LIN {X 89.707,Y 104.383,Z 77.424,A 180.000,B 0.000,C 180.000} C_DIS
LIN {X 89.757,Y 104.440,Z 77.421,A 180.000,B 0.000,C 180.000} C_DIS
LIN {X 89.860,Y 104.553,Z 77.416,A 180.000,B 0.000,C 180.000} C_DIS
LIN {X 90.120,Y 104.838,Z 77.402,A 180.000,B 0.000,C 180.000} C_DIS
LIN {X 90.174,Y 104.894,Z 77.400,A 180.000,B 0.000,C 180.000} C_DIS
LIN {X 90.229,Y 104.948,Z 77.397,A 180.000,B 0.000,C 180.000} C_DIS
LIN {X 90.451,Y 105.166,Z 77.386,A 180.000,B 0.000,C 180.000} C_DIS
LIN {X 90.507,Y 105.220,Z 77.383,A 180.000,B 0.000,C 180.000} C_DIS
LIN {X 90.564,Y 105.273,Z 77.381,A 180.000,B 0.000,C 180.000} C_DIS
LIN {X 90.622,Y 105.324,Z 77.378,A 180.000,B 0.000,C 180.000} C_DIS
LIN {X 90.855,Y 105.527,Z 77.367,A 180.000,B 0.000,C 180.000} C_DIS
LIN {X 90.914,Y 105.578,Z 77.364,A 180.000,B 0.000,C 180.000} C_DIS
LIN {X 90.973,Y 105.629,Z 77.362,A 180.000,B 0.000,C 180.000} C_DIS
LIN {X 91.033,Y 105.679,Z 77.359,A 180.000,B 0.000,C 180.000} C_DIS
LIN {X 91.093,Y 105.728,Z 77.356,A 180.000,B 0.000,C 180.000} C_DIS
LIN {X 91.397,Y 105.964,Z 77.343,A 180.000,B 0.000,C 180.000} C_DIS
LIN {X 91.458,Y 106.011,Z 77.340,A 180.000,B 0.000,C 180.000} C_DIS
LIN {X 91.521,Y 106.055,Z 77.337,A 180.000,B 0.000,C 180.000} C_DIS
LIN {X 91.650,Y 106.144,Z 77.332,A 180.000,B 0.000,C 180.000} C_DIS
LIN {X 91.779,Y 106.233,Z 77.326,A 180.000,B 0.000,C 180.000} C_DIS
LIN {X 91.843,Y 106.277,Z 77.324,A 180.000,B 0.000,C 180.000} C_DIS
LIN {X 91.907,Y 106.320,Z 77.321,A 180.000,B 0.000,C 180.000} C_DIS
LIN {X 91.972,Y 106.362,Z 77.318,A 180.000,B 0.000,C 180.000} C_DIS
LIN {X 92.036,Y 106.404,Z 77.316,A 180.000,B 0.000,C 180.000} C_DIS
LIN {X 92.103,Y 106.445,Z 77.313,A 180.000,B 0.000,C 180.000} C_DIS
LIN {X 92.236,Y 106.527,Z 77.307,A 180.000,B 0.000,C 180.000} C_DIS
LIN {X 92.303,Y 106.567,Z 77.305,A 180.000,B 0.000,C 180.000} C_DIS
LIN {X 92.369,Y 106.608,Z 77.302,A 180.000,B 0.000,C 180.000} C_DIS
LIN {X 92.434,Y 106.647,Z 77.299,A 180.000,B 0.000,C 180.000} C_DIS
LIN {X 92.501,Y 106.685,Z 77.297,A 180.000,B 0.000,C 180.000} C_DIS
LIN {X 92.569,Y 106.721,Z 77.294,A 180.000,B 0.000,C 180.000} C_DIS
LIN {X 92.707,Y 106.795,Z 77.289,A 180.000,B 0.000,C 180.000} C_DIS
LIN {X 92.845,Y 106.869,Z 77.283,A 180.000,B 0.000,C 180.000} C_DIS
LIN {X 92.914,Y 106.905,Z 77.280,A 180.000,B 0.000,C 180.000} C_DIS
LIN {X 92.983,Y 106.939,Z 77.278,A 180.000,B 0.000,C 180.000} C_DIS
LIN {X 93.053,Y 106.973,Z 77.275,A 180.000,B 0.000,C 180.000} C_DIS
LIN {X 93.123,Y 107.006,Z 77.272,A 180.000,B 0.000,C 180.000} C_DIS
LIN {X 93.266,Y 107.073,Z 77.267,A 180.000,B 0.000,C 180.000} C_DIS
LIN {X 93.408,Y 107.139,Z 77.261,A 180.000,B 0.000,C 180.000} C_DIS
LIN {X 93.478,Y 107.172,Z 77.259,A 180.000,B 0.000,C 180.000} C_DIS
LIN {X 93.549,Y 107.202,Z 77.256,A 180.000,B 0.000,C 180.000} C_DIS
LIN {X 93.620,Y 107.231,Z 77.253,A 180.000,B 0.000,C 180.000} C_DIS
LIN {X 93.692,Y 107.260,Z 77.250,A 180.000,B 0.000,C 180.000} C_DIS
LIN {X 93.837,Y 107.318,Z 77.245,A 180.000,B 0.000,C 180.000} C_DIS
LIN {X 93.909,Y 107.347,Z 77.242,A 180.000,B 0.000,C 180.000} C_DIS
LIN {X 93.982,Y 107.375,Z 77.240,A 180.000,B 0.000,C 180.000} C_DIS
LIN {X 94.055,Y 107.401,Z 77.237,A 180.000,B 0.000,C 180.000} C_DIS
LIN {X 94.129,Y 107.427,Z 77.234,A 180.000,B 0.000,C 180.000} C_DIS
LIN {X 94.203,Y 107.452,Z 77.231,A 180.000,B 0.000,C 180.000} C_DIS
LIN {X 94.277,Y 107.477,Z 77.229,A 180.000,B 0.000,C 180.000} C_DIS
LIN {X 94.426,Y 107.527,Z 77.223,A 180.000,B 0.000,C 180.000} C_DIS
LIN {X 94.500,Y 107.552,Z 77.220,A 180.000,B 0.000,C 180.000} C_DIS
LIN {X 94.575,Y 107.577,Z 77.218,A 180.000,B 0.000,C 180.000} C_DIS
LIN {X 94.649,Y 107.600,Z 77.215,A 180.000,B 0.000,C 180.000} C_DIS
LIN {X 94.723,Y 107.621,Z 77.212,A 180.000,B 0.000,C 180.000} C_DIS
LIN {X 94.947,Y 107.683,Z 77.204,A 180.000,B 0.000,C 180.000} C_DIS
LIN {X 95.022,Y 107.704,Z 77.201,A 180.000,B 0.000,C 180.000} C_DIS
LIN {X 95.097,Y 107.724,Z 77.199,A 180.000,B 0.000,C 180.000} C_DIS
LIN {X 95.173,Y 107.742,Z 77.196,A 180.000,B 0.000,C 180.000} C_DIS
LIN {X 95.249,Y 107.759,Z 77.193,A 180.000,B 0.000,C 180.000} C_DIS
LIN {X 95.326,Y 107.776,Z 77.191,A 180.000,B 0.000,C 180.000} C_DIS
LIN {X 95.403,Y 107.792,Z 77.188,A 180.000,B 0.000,C 180.000} C_DIS
LIN {X 95.480,Y 107.809,Z 77.185,A 180.000,B 0.000,C 180.000} C_DIS
LIN {X 95.556,Y 107.825,Z 77.182,A 180.000,B 0.000,C 180.000} C_DIS
LIN {X 95.633,Y 107.842,Z 77.180,A 180.000,B 0.000,C 180.000} C_DIS
LIN {X 95.710,Y 107.858,Z 77.177,A 180.000,B 0.000,C 180.000} C_DIS
LIN {X 95.787,Y 107.873,Z 77.174,A 180.000,B 0.000,C 180.000} C_DIS
LIN {X 95.864,Y 107.886,Z 77.172,A 180.000,B 0.000,C 180.000} C_DIS
LIN {X 95.941,Y 107.898,Z 77.169,A 180.000,B 0.000,C 180.000} C_DIS
LIN {X 96.018,Y 107.910,Z 77.167,A 180.000,B 0.000,C 180.000} C_DIS
LIN {X 96.095,Y 107.922,Z 77.164,A 180.000,B 0.000,C 180.000} C_DIS
LIN {X 96.172,Y 107.934,Z 77.162,A 180.000,B 0.000,C 180.000} C_DIS
LIN {X 96.248,Y 107.946,Z 77.159,A 180.000,B 0.000,C 180.000} C_DIS
LIN {X 96.325,Y 107.957,Z 77.156,A 180.000,B 0.000,C 180.000} C_DIS
LIN {X 96.403,Y 107.965,Z 77.154,A 180.000,B 0.000,C 180.000} C_DIS
LIN {X 96.481,Y 107.973,Z 77.151,A 180.000,B 0.000,C 180.000} C_DIS
LIN {X 96.560,Y 107.981,Z 77.149,A 180.000,B 0.000,C 180.000} C_DIS
LIN {X 96.716,Y 107.996,Z 77.144,A 180.000,B 0.000,C 180.000} C_DIS
LIN {X 96.872,Y 108.010,Z 77.139,A 180.000,B 0.000,C 180.000} C_DIS
LIN {X 97.028,Y 108.021,Z 77.134,A 180.000,B 0.000,C 180.000} C_DIS
LIN {X 97.185,Y 108.027,Z 77.130,A 180.000,B 0.000,C 180.000} C_DIS
LIN {X 97.341,Y 108.034,Z 77.125,A 180.000,B 0.000,C 180.000} C_DIS
LIN {X 97.497,Y 108.040,Z 77.120,A 180.000,B 0.000,C 180.000} C_DIS
LIN {X 97.653,Y 108.038,Z 77.116,A 180.000,B 0.000,C 180.000} C_DIS
LIN {X 97.810,Y 108.036,Z 77.111,A 180.000,B 0.000,C 180.000} C_DIS
LIN {X 97.968,Y 108.034,Z 77.107,A 180.000,B 0.000,C 180.000} C_DIS
LIN {X 98.124,Y 108.027,Z 77.102,A 180.000,B 0.000,C 180.000} C_DIS
LIN {X 98.281,Y 108.018,Z 77.098,A 180.000,B 0.000,C 180.000} C_DIS
LIN {X 98.437,Y 108.007,Z 77.094,A 180.000,B 0.000,C 180.000} C_DIS
LIN {X 98.594,Y 107.995,Z 77.090,A 180.000,B 0.000,C 180.000} C_DIS
LIN {X 98.750,Y 107.981,Z 77.086,A 180.000,B 0.000,C 180.000} C_DIS
LIN {X 98.905,Y 107.961,Z 77.082,A 180.000,B 0.000,C 180.000} C_DIS
LIN {X 99.061,Y 107.941,Z 77.078,A 180.000,B 0.000,C 180.000} C_DIS
LIN {X 99.216,Y 107.920,Z 77.074,A 180.000,B 0.000,C 180.000} C_DIS
LIN {X 99.371,Y 107.893,Z 77.071,A 180.000,B 0.000,C 180.000} C_DIS
LIN {X 99.526,Y 107.864,Z 77.067,A 180.000,B 0.000,C 180.000} C_DIS
LIN {X 99.680,Y 107.835,Z 77.063,A 180.000,B 0.000,C 180.000} C_DIS
LIN {X 99.835,Y 107.806,Z 77.060,A 180.000,B 0.000,C 180.000} C_DIS
LIN {X 99.988,Y 107.771,Z 77.056,A 180.000,B 0.000,C 180.000} C_DIS
LIN {X 100.140,Y 107.733,Z 77.053,A 180.000,B 0.000,C 180.000} C_DIS
LIN {X 100.293,Y 107.695,Z 77.050,A 180.000,B 0.000,C 180.000} C_DIS
LIN {X 100.445,Y 107.655,Z 77.047,A 180.000,B 0.000,C 180.000} C_DIS
LIN {X 100.595,Y 107.608,Z 77.044,A 180.000,B 0.000,C 180.000} C_DIS
LIN {X 100.745,Y 107.562,Z 77.041,A 180.000,B 0.000,C 180.000} C_DIS
LIN {X 100.895,Y 107.515,Z 77.038,A 180.000,B 0.000,C 180.000} C_DIS
LIN {X 101.045,Y 107.467,Z 77.035,A 180.000,B 0.000,C 180.000} C_DIS
LIN {X 101.192,Y 107.413,Z 77.033,A 180.000,B 0.000,C 180.000} C_DIS
LIN {X 101.340,Y 107.358,Z 77.030,A 180.000,B 0.000,C 180.000} C_DIS
LIN {X 101.632,Y 107.242,Z 77.025,A 180.000,B 0.000,C 180.000} C_DIS
LIN {X 101.920,Y 107.115,Z 77.021,A 180.000,B 0.000,C 180.000} C_DIS
LIN {X 102.206,Y 106.983,Z 77.017,A 180.000,B 0.000,C 180.000} C_DIS
LIN {X 102.486,Y 106.840,Z 77.013,A 180.000,B 0.000,C 180.000} C_DIS
LIN {X 102.762,Y 106.689,Z 77.010,A 180.000,B 0.000,C 180.000} C_DIS
LIN {X 103.034,Y 106.530,Z 77.007,A 180.000,B 0.000,C 180.000} C_DIS
LIN {X 103.300,Y 106.361,Z 77.005,A 180.000,B 0.000,C 180.000} C_DIS
LIN {X 103.562,Y 106.187,Z 77.003,A 180.000,B 0.000,C 180.000} C_DIS
LIN {X 103.817,Y 106.002,Z 77.001,A 180.000,B 0.000,C 180.000} C_DIS
LIN {X 104.069,Y 105.812,Z 77.001,A 180.000,B 0.000,C 180.000} C_DIS
LIN {X 104.311,Y 105.611,Z 77.000,A 180.000,B 0.000,C 180.000} C_DIS
LIN {X 104.414,Y 105.524,Z 77.000,A 180.000,B 0.000,C 180.000} C_DIS
; Cutting Move Starts
LIN {X 104.469,Y 105.477,Z 77.000,A 180.000,B 0.000,C 180.000} C_DIS
LIN {X 104.584,Y 105.379,Z 77.000,A 180.000,B 0.000,C 180.000} C_DIS
LIN {X 104.670,Y 105.299,Z 77.000,A 180.000,B 0.000,C 180.000} C_DIS
LIN {X 104.859,Y 105.120,Z 77.000,A 180.000,B 0.000,C 180.000} C_DIS
LIN {X 104.941,Y 105.042,Z 77.000,A 180.000,B 0.000,C 180.000} C_DIS
LIN {X 105.040,Y 104.941,Z 77.000,A 180.000,B 0.000,C 180.000} C_DIS
LIN {X 105.209,Y 104.762,Z 77.000,A 180.000,B 0.000,C 180.000} C_DIS
LIN {X 105.299,Y 104.667,Z 77.000,A 180.000,B 0.000,C 180.000} C_DIS
LIN {X 105.377,Y 104.584,Z 77.000,A 180.000,B 0.000,C 180.000} C_DIS
LIN {X 105.477,Y 104.471,Z 77.000,A 180.000,B 0.000,C 180.000} C_DIS
LIN {X 105.685,Y 104.226,Z 77.000,A 180.000,B 0.000,C 180.000} C_DIS
LIN {X 105.829,Y 104.047,Z 77.000,A 180.000,B 0.000,C 180.000} C_DIS
LIN {X 106.014,Y 103.801,Z 77.000,A 180.000,B 0.000,C 180.000} C_DIS
LIN {X 106.097,Y 103.690,Z 77.000,A 180.000,B 0.000,C 180.000} C_DIS
LIN {X 106.193,Y 103.556,Z 77.000,A 180.000,B 0.000,C 180.000} C_DIS
LIN {X 106.223,Y 103.511,Z 77.000,A 180.000,B 0.000,C 180.000} C_DIS
LIN {X 106.371,Y 103.289,Z 77.000,A 180.000,B 0.000,C 180.000} C_DIS
LIN {X 106.461,Y 103.153,Z 77.000,A 180.000,B 0.000,C 180.000} C_DIS
LIN {X 106.550,Y 103.006,Z 77.000,A 180.000,B 0.000,C 180.000} C_DIS
LIN {X 106.674,Y 102.796,Z 77.000,A 180.000,B 0.000,C 180.000} C_DIS
LIN {X 106.729,Y 102.702,Z 77.000,A 180.000,B 0.000,C 180.000} C_DIS
LIN {X 106.776,Y 102.617,Z 77.000,A 180.000,B 0.000,C 180.000} C_DIS
LIN {X 106.871,Y 102.438,Z 77.000,A 180.000,B 0.000,C 180.000} C_DIS
LIN {X 106.963,Y 102.260,Z 77.000,A 180.000,B 0.000,C 180.000} C_DIS
LIN {X 107.054,Y 102.081,Z 77.000,A 180.000,B 0.000,C 180.000} C_DIS
LIN {X 107.086,Y 102.011,Z 77.000,A 180.000,B 0.000,C 180.000} C_DIS
LIN {X 107.215,Y 101.723,Z 77.000,A 180.000,B 0.000,C 180.000} C_DIS
LIN {X 107.265,Y 101.609,Z 77.000,A 180.000,B 0.000,C 180.000} C_DIS
LIN {X 107.291,Y 101.545,Z 77.000,A 180.000,B 0.000,C 180.000} C_DIS
LIN {X 107.361,Y 101.366,Z 77.000,A 180.000,B 0.000,C 180.000} C_DIS
LIN {X 107.444,Y 101.149,Z 77.000,A 180.000,B 0.000,C 180.000} C_DIS
LIN {X 107.498,Y 101.008,Z 77.000,A 180.000,B 0.000,C 180.000} C_DIS
LIN {X 107.557,Y 100.829,Z 77.000,A 180.000,B 0.000,C 180.000} C_DIS
LIN {X 107.623,Y 100.623,Z 77.000,A 180.000,B 0.000,C 180.000} C_DIS
LIN {X 107.670,Y 100.472,Z 77.000,A 180.000,B 0.000,C 180.000} C_DIS
LIN {X 107.717,Y 100.293,Z 77.000,A 180.000,B 0.000,C 180.000} C_DIS
LIN {X 107.763,Y 100.114,Z 77.000,A 180.000,B 0.000,C 180.000} C_DIS
LIN {X 107.802,Y 99.965,Z 77.000,A 180.000,B 0.000,C 180.000} C_DIS
LIN {X 107.809,Y 99.936,Z 77.000,A 180.000,B 0.000,C 180.000} C_DIS
LIN {X 107.852,Y 99.757,Z 77.000,A 180.000,B 0.000,C 180.000} C_DIS
LIN {X 107.923,Y 99.399,Z 77.000,A 180.000,B 0.000,C 180.000} C_DIS
LIN {X 107.954,Y 99.221,Z 77.000,A 180.000,B 0.000,C 180.000} C_DIS
LIN {X 108.004,Y 98.863,Z 77.000,A 180.000,B 0.000,C 180.000} C_DIS
LIN {X 108.027,Y 98.684,Z 77.000,A 180.000,B 0.000,C 180.000} C_DIS
LIN {X 108.045,Y 98.505,Z 77.000,A 180.000,B 0.000,C 180.000} C_DIS
LIN {X 108.061,Y 98.327,Z 77.000,A 180.000,B 0.000,C 180.000} C_DIS
LIN {X 108.076,Y 98.148,Z 77.000,A 180.000,B 0.000,C 180.000} C_DIS
LIN {X 108.083,Y 97.969,Z 77.000,A 180.000,B 0.000,C 180.000} C_DIS
LIN {X 108.088,Y 97.790,Z 77.000,A 180.000,B 0.000,C 180.000} C_DIS
LIN {X 108.093,Y 97.612,Z 77.000,A 180.000,B 0.000,C 180.000} C_DIS
LIN {X 108.094,Y 97.433,Z 77.000,A 180.000,B 0.000,C 180.000} C_DIS
LIN {X 108.090,Y 97.254,Z 77.000,A 180.000,B 0.000,C 180.000} C_DIS
LIN {X 108.085,Y 97.075,Z 77.000,A 180.000,B 0.000,C 180.000} C_DIS
LIN {X 108.078,Y 96.897,Z 77.000,A 180.000,B 0.000,C 180.000} C_DIS
LIN {X 108.064,Y 96.718,Z 77.000,A 180.000,B 0.000,C 180.000} C_DIS
LIN {X 108.049,Y 96.539,Z 77.000,A 180.000,B 0.000,C 180.000} C_DIS
LIN {X 108.033,Y 96.360,Z 77.000,A 180.000,B 0.000,C 180.000} C_DIS
LIN {X 108.010,Y 96.181,Z 77.000,A 180.000,B 0.000,C 180.000} C_DIS
LIN {X 107.985,Y 96.003,Z 77.000,A 180.000,B 0.000,C 180.000} C_DIS
LIN {X 107.960,Y 95.824,Z 77.000,A 180.000,B 0.000,C 180.000} C_DIS
LIN {X 107.931,Y 95.645,Z 77.000,A 180.000,B 0.000,C 180.000} C_DIS
LIN {X 107.896,Y 95.466,Z 77.000,A 180.000,B 0.000,C 180.000} C_DIS
LIN {X 107.860,Y 95.288,Z 77.000,A 180.000,B 0.000,C 180.000} C_DIS
LIN {X 107.821,Y 95.109,Z 77.000,A 180.000,B 0.000,C 180.000} C_DIS
LIN {X 107.802,Y 95.035,Z 77.000,A 180.000,B 0.000,C 180.000} C_DIS
LIN {X 107.775,Y 94.930,Z 77.000,A 180.000,B 0.000,C 180.000} C_DIS
LIN {X 107.728,Y 94.751,Z 77.000,A 180.000,B 0.000,C 180.000} C_DIS
LIN {X 107.682,Y 94.573,Z 77.000,A 180.000,B 0.000,C 180.000} C_DIS
LIN {X 107.628,Y 94.394,Z 77.000,A 180.000,B 0.000,C 180.000} C_DIS
LIN {X 107.571,Y 94.215,Z 77.000,A 180.000,B 0.000,C 180.000} C_DIS
LIN {X 107.513,Y 94.036,Z 77.000,A 180.000,B 0.000,C 180.000} C_DIS
LIN {X 107.447,Y 93.857,Z 77.000,A 180.000,B 0.000,C 180.000} C_DIS
LIN {X 107.378,Y 93.679,Z 77.000,A 180.000,B 0.000,C 180.000} C_DIS
LIN {X 107.309,Y 93.500,Z 77.000,A 180.000,B 0.000,C 180.000} C_DIS
LIN {X 107.265,Y 93.391,Z 77.000,A 180.000,B 0.000,C 180.000} C_DIS
LIN {X 107.235,Y 93.321,Z 77.000,A 180.000,B 0.000,C 180.000} C_DIS
LIN {X 107.086,Y 92.989,Z 77.000,A 180.000,B 0.000,C 180.000} C_DIS
LIN {X 107.075,Y 92.964,Z 77.000,A 180.000,B 0.000,C 180.000} C_DIS
LIN {X 106.986,Y 92.785,Z 77.000,A 180.000,B 0.000,C 180.000} C_DIS
LIN {X 106.894,Y 92.606,Z 77.000,A 180.000,B 0.000,C 180.000} C_DIS
LIN {X 106.800,Y 92.427,Z 77.000,A 180.000,B 0.000,C 180.000} C_DIS
LIN {X 106.729,Y 92.298,Z 77.000,A 180.000,B 0.000,C 180.000} C_DIS
LIN {X 106.700,Y 92.249,Z 77.000,A 180.000,B 0.000,C 180.000} C_DIS
LIN {X 106.550,Y 91.994,Z 77.000,A 180.000,B 0.000,C 180.000} C_DIS
LIN {X 106.489,Y 91.891,Z 77.000,A 180.000,B 0.000,C 180.000} C_DIS
LIN {X 106.372,Y 91.712,Z 77.000,A 180.000,B 0.000,C 180.000} C_DIS
LIN {X 106.253,Y 91.533,Z 77.000,A 180.000,B 0.000,C 180.000} C_DIS
LIN {X 106.193,Y 91.444,Z 77.000,A 180.000,B 0.000,C 180.000} C_DIS
LIN {X 106.129,Y 91.355,Z 77.000,A 180.000,B 0.000,C 180.000} C_DIS
LIN {X 106.014,Y 91.199,Z 77.000,A 180.000,B 0.000,C 180.000} C_DIS
LIN {X 105.835,Y 90.961,Z 77.000,A 180.000,B 0.000,C 180.000} C_DIS
LIN {X 105.722,Y 90.818,Z 77.000,A 180.000,B 0.000,C 180.000} C_DIS
LIN {X 105.477,Y 90.529,Z 77.000,A 180.000,B 0.000,C 180.000} C_DIS
LIN {X 105.418,Y 90.461,Z 77.000,A 180.000,B 0.000,C 180.000} C_DIS
LIN {X 105.299,Y 90.333,Z 77.000,A 180.000,B 0.000,C 180.000} C_DIS
LIN {X 105.251,Y 90.282,Z 77.000,A 180.000,B 0.000,C 180.000} C_DIS
LIN {X 105.082,Y 90.103,Z 77.000,A 180.000,B 0.000,C 180.000} C_DIS
LIN {X 104.941,Y 89.958,Z 77.000,A 180.000,B 0.000,C 180.000} C_DIS
LIN {X 104.906,Y 89.925,Z 77.000,A 180.000,B 0.000,C 180.000} C_DIS
LIN {X 104.717,Y 89.746,Z 77.000,A 180.000,B 0.000,C 180.000} C_DIS
LIN {X 104.584,Y 89.621,Z 77.000,A 180.000,B 0.000,C 180.000} C_DIS
LIN {X 104.522,Y 89.567,Z 77.000,A 180.000,B 0.000,C 180.000} C_DIS
LIN {X 104.226,Y 89.317,Z 77.000,A 180.000,B 0.000,C 180.000} C_DIS
LIN {X 104.096,Y 89.209,Z 77.000,A 180.000,B 0.000,C 180.000} C_DIS
LIN {X 104.047,Y 89.171,Z 77.000,A 180.000,B 0.000,C 180.000} C_DIS
LIN {X 103.869,Y 89.035,Z 77.000,A 180.000,B 0.000,C 180.000} C_DIS
LIN {X 103.690,Y 88.901,Z 77.000,A 180.000,B 0.000,C 180.000} C_DIS
LIN {X 103.622,Y 88.852,Z 77.000,A 180.000,B 0.000,C 180.000} C_DIS
LIN {X 103.511,Y 88.777,Z 77.000,A 180.000,B 0.000,C 180.000} C_DIS
LIN {X 103.332,Y 88.658,Z 77.000,A 180.000,B 0.000,C 180.000} C_DIS
LIN {X 103.153,Y 88.541,Z 77.000,A 180.000,B 0.000,C 180.000} C_DIS
LIN {X 103.080,Y 88.494,Z 77.000,A 180.000,B 0.000,C 180.000} C_DIS
LIN {X 102.975,Y 88.431,Z 77.000,A 180.000,B 0.000,C 180.000} C_DIS
LIN {X 102.778,Y 88.316,Z 77.000,A 180.000,B 0.000,C 180.000} C_DIS
LIN {X 102.617,Y 88.222,Z 77.000,A 180.000,B 0.000,C 180.000} C_DIS
LIN {X 102.454,Y 88.137,Z 77.000,A 180.000,B 0.000,C 180.000} C_DIS
LIN {X 102.260,Y 88.036,Z 77.000,A 180.000,B 0.000,C 180.000} C_DIS
LIN {X 102.102,Y 87.958,Z 77.000,A 180.000,B 0.000,C 180.000} C_DIS
LIN {X 102.081,Y 87.948,Z 77.000,A 180.000,B 0.000,C 180.000} C_DIS
LIN {X 101.902,Y 87.866,Z 77.000,A 180.000,B 0.000,C 180.000} C_DIS
LIN {X 101.709,Y 87.779,Z 77.000,A 180.000,B 0.000,C 180.000} C_DIS
LIN {X 101.545,Y 87.707,Z 77.000,A 180.000,B 0.000,C 180.000} C_DIS
LIN {X 101.366,Y 87.637,Z 77.000,A 180.000,B 0.000,C 180.000} C_DIS
LIN {X 101.187,Y 87.569,Z 77.000,A 180.000,B 0.000,C 180.000} C_DIS
LIN {X 101.008,Y 87.503,Z 77.000,A 180.000,B 0.000,C 180.000} C_DIS
LIN {X 100.829,Y 87.445,Z 77.000,A 180.000,B 0.000,C 180.000} C_DIS
LIN {X 100.472,Y 87.331,Z 77.000,A 180.000,B 0.000,C 180.000} C_DIS
LIN {X 100.293,Y 87.281,Z 77.000,A 180.000,B 0.000,C 180.000} C_DIS
LIN {X 100.114,Y 87.235,Z 77.000,A 180.000,B 0.000,C 180.000} C_DIS
LIN {X 99.936,Y 87.189,Z 77.000,A 180.000,B 0.000,C 180.000} C_DIS
LIN {X 99.757,Y 87.150,Z 77.000,A 180.000,B 0.000,C 180.000} C_DIS
LIN {X 99.578,Y 87.115,Z 77.000,A 180.000,B 0.000,C 180.000} C_DIS
LIN {X 99.399,Y 87.079,Z 77.000,A 180.000,B 0.000,C 180.000} C_DIS
LIN {X 99.321,Y 87.064,Z 77.000,A 180.000,B 0.000,C 180.000} C_DIS
LIN {X 99.221,Y 87.046,Z 77.000,A 180.000,B 0.000,C 180.000} C_DIS
LIN {X 99.042,Y 87.020,Z 77.000,A 180.000,B 0.000,C 180.000} C_DIS
LIN {X 98.863,Y 86.995,Z 77.000,A 180.000,B 0.000,C 180.000} C_DIS
LIN {X 98.684,Y 86.971,Z 77.000,A 180.000,B 0.000,C 180.000} C_DIS
LIN {X 98.505,Y 86.955,Z 77.000,A 180.000,B 0.000,C 180.000} C_DIS
LIN {X 98.327,Y 86.940,Z 77.000,A 180.000,B 0.000,C 180.000} C_DIS
LIN {X 98.148,Y 86.926,Z 77.000,A 180.000,B 0.000,C 180.000} C_DIS
LIN {X 97.969,Y 86.916,Z 77.000,A 180.000,B 0.000,C 180.000} C_DIS
LIN {X 97.612,Y 86.906,Z 77.000,A 180.000,B 0.000,C 180.000} C_DIS
LIN {X 97.433,Y 86.905,Z 77.000,A 180.000,B 0.000,C 180.000} C_DIS
LIN {X 97.075,Y 86.915,Z 77.000,A 180.000,B 0.000,C 180.000} C_DIS
LIN {X 96.897,Y 86.924,Z 77.000,A 180.000,B 0.000,C 180.000} C_DIS
LIN {X 96.718,Y 86.936,Z 77.000,A 180.000,B 0.000,C 180.000} C_DIS
LIN {X 96.539,Y 86.951,Z 77.000,A 180.000,B 0.000,C 180.000} C_DIS
LIN {X 96.360,Y 86.967,Z 77.000,A 180.000,B 0.000,C 180.000} C_DIS
LIN {X 96.181,Y 86.988,Z 77.000,A 180.000,B 0.000,C 180.000} C_DIS
LIN {X 96.003,Y 87.014,Z 77.000,A 180.000,B 0.000,C 180.000} C_DIS
LIN {X 95.824,Y 87.039,Z 77.000,A 180.000,B 0.000,C 180.000} C_DIS
LIN {X 95.679,Y 87.064,Z 77.000,A 180.000,B 0.000,C 180.000} C_DIS
LIN {X 95.645,Y 87.071,Z 77.000,A 180.000,B 0.000,C 180.000} C_DIS
LIN {X 95.466,Y 87.106,Z 77.000,A 180.000,B 0.000,C 180.000} C_DIS
LIN {X 95.288,Y 87.141,Z 77.000,A 180.000,B 0.000,C 180.000} C_DIS
LIN {X 95.109,Y 87.178,Z 77.000,A 180.000,B 0.000,C 180.000} C_DIS
LIN {X 94.930,Y 87.223,Z 77.000,A 180.000,B 0.000,C 180.000} C_DIS
LIN {X 94.751,Y 87.269,Z 77.000,A 180.000,B 0.000,C 180.000} C_DIS
LIN {X 94.654,Y 87.295,Z 77.000,A 180.000,B 0.000,C 180.000} C_DIS
LIN {X 94.573,Y 87.317,Z 77.000,A 180.000,B 0.000,C 180.000} C_DIS
LIN {X 94.394,Y 87.374,Z 77.000,A 180.000,B 0.000,C 180.000} C_DIS
LIN {X 94.215,Y 87.431,Z 77.000,A 180.000,B 0.000,C 180.000} C_DIS
LIN {X 94.036,Y 87.489,Z 77.000,A 180.000,B 0.000,C 180.000} C_DIS
LIN {X 93.857,Y 87.552,Z 77.000,A 180.000,B 0.000,C 180.000} C_DIS
LIN {X 93.679,Y 87.620,Z 77.000,A 180.000,B 0.000,C 180.000} C_DIS
LIN {X 93.500,Y 87.689,Z 77.000,A 180.000,B 0.000,C 180.000} C_DIS
LIN {X 93.321,Y 87.766,Z 77.000,A 180.000,B 0.000,C 180.000} C_DIS
LIN {X 93.142,Y 87.846,Z 77.000,A 180.000,B 0.000,C 180.000} C_DIS
LIN {X 92.964,Y 87.927,Z 77.000,A 180.000,B 0.000,C 180.000} C_DIS
LIN {X 92.898,Y 87.958,Z 77.000,A 180.000,B 0.000,C 180.000} C_DIS
LIN {X 92.785,Y 88.013,Z 77.000,A 180.000,B 0.000,C 180.000} C_DIS
LIN {X 92.546,Y 88.137,Z 77.000,A 180.000,B 0.000,C 180.000} C_DIS
LIN {X 92.427,Y 88.198,Z 77.000,A 180.000,B 0.000,C 180.000} C_DIS
LIN {X 92.249,Y 88.300,Z 77.000,A 180.000,B 0.000,C 180.000} C_DIS
LIN {X 92.070,Y 88.405,Z 77.000,A 180.000,B 0.000,C 180.000} C_DIS
LIN {X 91.920,Y 88.494,Z 77.000,A 180.000,B 0.000,C 180.000} C_DIS
LIN {X 91.891,Y 88.513,Z 77.000,A 180.000,B 0.000,C 180.000} C_DIS
LIN {X 91.712,Y 88.628,Z 77.000,A 180.000,B 0.000,C 180.000} C_DIS
LIN {X 91.533,Y 88.748,Z 77.000,A 180.000,B 0.000,C 180.000} C_DIS
LIN {X 91.378,Y 88.852,Z 77.000,A 180.000,B 0.000,C 180.000} C_DIS
LIN {X 91.355,Y 88.869,Z 77.000,A 180.000,B 0.000,C 180.000} C_DIS
LIN {X 91.176,Y 89.002,Z 77.000,A 180.000,B 0.000,C 180.000} C_DIS
LIN {X 90.997,Y 89.137,Z 77.000,A 180.000,B 0.000,C 180.000} C_DIS
LIN {X 90.904,Y 89.209,Z 77.000,A 180.000,B 0.000,C 180.000} C_DIS
LIN {X 90.818,Y 89.280,Z 77.000,A 180.000,B 0.000,C 180.000} C_DIS
LIN {X 90.690,Y 89.388,Z 77.000,A 180.000,B 0.000,C 180.000} C_DIS
LIN {X 90.478,Y 89.567,Z 77.000,A 180.000,B 0.000,C 180.000} C_DIS
LIN {X 90.461,Y 89.582,Z 77.000,A 180.000,B 0.000,C 180.000} C_DIS
LIN {X 90.283,Y 89.746,Z 77.000,A 180.000,B 0.000,C 180.000} C_DIS
LIN {X 90.094,Y 89.925,Z 77.000,A 180.000,B 0.000,C 180.000} C_DIS
LIN {X 89.925,Y 90.096,Z 77.000,A 180.000,B 0.000,C 180.000} C_DIS
LIN {X 89.746,Y 90.286,Z 77.000,A 180.000,B 0.000,C 180.000} C_DIS
LIN {X 89.582,Y 90.461,Z 77.000,A 180.000,B 0.000,C 180.000} C_DIS
LIN {X 89.567,Y 90.477,Z 77.000,A 180.000,B 0.000,C 180.000} C_DIS
LIN {X 89.429,Y 90.640,Z 77.000,A 180.000,B 0.000,C 180.000} C_DIS
LIN {X 89.278,Y 90.818,Z 77.000,A 180.000,B 0.000,C 180.000} C_DIS
LIN {X 89.209,Y 90.902,Z 77.000,A 180.000,B 0.000,C 180.000} C_DIS
LIN {X 89.138,Y 90.997,Z 77.000,A 180.000,B 0.000,C 180.000} C_DIS
LIN {X 89.003,Y 91.176,Z 77.000,A 180.000,B 0.000,C 180.000} C_DIS
LIN {X 88.871,Y 91.355,Z 77.000,A 180.000,B 0.000,C 180.000} C_DIS
LIN {X 88.852,Y 91.381,Z 77.000,A 180.000,B 0.000,C 180.000} C_DIS
LIN {X 88.747,Y 91.533,Z 77.000,A 180.000,B 0.000,C 180.000} C_DIS
LIN {X 88.628,Y 91.712,Z 77.000,A 180.000,B 0.000,C 180.000} C_DIS
LIN {X 88.511,Y 91.891,Z 77.000,A 180.000,B 0.000,C 180.000} C_DIS
LIN {X 88.494,Y 91.919,Z 77.000,A 180.000,B 0.000,C 180.000} C_DIS
LIN {X 88.300,Y 92.249,Z 77.000,A 180.000,B 0.000,C 180.000} C_DIS
LIN {X 88.200,Y 92.427,Z 77.000,A 180.000,B 0.000,C 180.000} C_DIS
LIN {X 88.137,Y 92.547,Z 77.000,A 180.000,B 0.000,C 180.000} C_DIS
LIN {X 88.014,Y 92.785,Z 77.000,A 180.000,B 0.000,C 180.000} C_DIS
LIN {X 87.958,Y 92.894,Z 77.000,A 180.000,B 0.000,C 180.000} C_DIS
LIN {X 87.925,Y 92.964,Z 77.000,A 180.000,B 0.000,C 180.000} C_DIS
LIN {X 87.845,Y 93.142,Z 77.000,A 180.000,B 0.000,C 180.000} C_DIS
LIN {X 87.765,Y 93.321,Z 77.000,A 180.000,B 0.000,C 180.000} C_DIS
LIN {X 87.691,Y 93.500,Z 77.000,A 180.000,B 0.000,C 180.000} C_DIS
LIN {X 87.622,Y 93.679,Z 77.000,A 180.000,B 0.000,C 180.000} C_DIS
LIN {X 87.553,Y 93.857,Z 77.000,A 180.000,B 0.000,C 180.000} C_DIS
LIN {X 87.487,Y 94.036,Z 77.000,A 180.000,B 0.000,C 180.000} C_DIS
LIN {X 87.429,Y 94.215,Z 77.000,A 180.000,B 0.000,C 180.000} C_DIS
LIN {X 87.372,Y 94.394,Z 77.000,A 180.000,B 0.000,C 180.000} C_DIS
LIN {X 87.318,Y 94.573,Z 77.000,A 180.000,B 0.000,C 180.000} C_DIS
LIN {X 87.272,Y 94.751,Z 77.000,A 180.000,B 0.000,C 180.000} C_DIS
LIN {X 87.225,Y 94.930,Z 77.000,A 180.000,B 0.000,C 180.000} C_DIS
LIN {X 87.179,Y 95.109,Z 77.000,A 180.000,B 0.000,C 180.000} C_DIS
LIN {X 87.140,Y 95.288,Z 77.000,A 180.000,B 0.000,C 180.000} C_DIS
LIN {X 87.104,Y 95.466,Z 77.000,A 180.000,B 0.000,C 180.000} C_DIS
LIN {X 87.069,Y 95.645,Z 77.000,A 180.000,B 0.000,C 180.000} C_DIS
LIN {X 87.064,Y 95.668,Z 77.000,A 180.000,B 0.000,C 180.000} C_DIS
LIN {X 87.040,Y 95.824,Z 77.000,A 180.000,B 0.000,C 180.000} C_DIS
LIN {X 87.015,Y 96.003,Z 77.000,A 180.000,B 0.000,C 180.000} C_DIS
LIN {X 86.990,Y 96.181,Z 77.000,A 180.000,B 0.000,C 180.000} C_DIS
LIN {X 86.977,Y 96.280,Z 77.000,A 180.000,B 0.000,C 180.000} C_DIS
LIN {X 86.967,Y 96.360,Z 77.000,A 180.000,B 0.000,C 180.000} C_DIS
LIN {X 86.951,Y 96.539,Z 77.000,A 180.000,B 0.000,C 180.000} C_DIS
LIN {X 86.936,Y 96.718,Z 77.000,A 180.000,B 0.000,C 180.000} C_DIS
LIN {X 86.922,Y 96.897,Z 77.000,A 180.000,B 0.000,C 180.000} C_DIS
LIN {X 86.915,Y 97.075,Z 77.000,A 180.000,B 0.000,C 180.000} C_DIS
LIN {X 86.910,Y 97.254,Z 77.000,A 180.000,B 0.000,C 180.000} C_DIS
LIN {X 86.906,Y 97.433,Z 77.000,A 180.000,B 0.000,C 180.000} C_DIS
LIN {X 86.907,Y 97.612,Z 77.000,A 180.000,B 0.000,C 180.000} C_DIS
LIN {X 86.912,Y 97.790,Z 77.000,A 180.000,B 0.000,C 180.000} C_DIS
LIN {X 86.917,Y 97.969,Z 77.000,A 180.000,B 0.000,C 180.000} C_DIS
LIN {X 86.924,Y 98.148,Z 77.000,A 180.000,B 0.000,C 180.000} C_DIS
LIN {X 86.939,Y 98.327,Z 77.000,A 180.000,B 0.000,C 180.000} C_DIS
LIN {X 86.955,Y 98.505,Z 77.000,A 180.000,B 0.000,C 180.000} C_DIS
LIN {X 86.973,Y 98.684,Z 77.000,A 180.000,B 0.000,C 180.000} C_DIS
LIN {X 86.996,Y 98.863,Z 77.000,A 180.000,B 0.000,C 180.000} C_DIS
LIN {X 87.046,Y 99.221,Z 77.000,A 180.000,B 0.000,C 180.000} C_DIS
LIN {X 87.064,Y 99.332,Z 77.000,A 180.000,B 0.000,C 180.000} C_DIS
LIN {X 87.077,Y 99.399,Z 77.000,A 180.000,B 0.000,C 180.000} C_DIS
LIN {X 87.148,Y 99.757,Z 77.000,A 180.000,B 0.000,C 180.000} C_DIS
LIN {X 87.191,Y 99.936,Z 77.000,A 180.000,B 0.000,C 180.000} C_DIS
LIN {X 87.237,Y 100.114,Z 77.000,A 180.000,B 0.000,C 180.000} C_DIS
LIN {X 87.283,Y 100.293,Z 77.000,A 180.000,B 0.000,C 180.000} C_DIS
LIN {X 87.330,Y 100.472,Z 77.000,A 180.000,B 0.000,C 180.000} C_DIS
LIN {X 87.386,Y 100.651,Z 77.000,A 180.000,B 0.000,C 180.000} C_DIS
LIN {X 87.443,Y 100.829,Z 77.000,A 180.000,B 0.000,C 180.000} C_DIS
LIN {X 87.502,Y 101.008,Z 77.000,A 180.000,B 0.000,C 180.000} C_DIS
LIN {X 87.570,Y 101.187,Z 77.000,A 180.000,B 0.000,C 180.000} C_DIS
LIN {X 87.639,Y 101.366,Z 77.000,A 180.000,B 0.000,C 180.000} C_DIS
LIN {X 87.709,Y 101.545,Z 77.000,A 180.000,B 0.000,C 180.000} C_DIS
LIN {X 87.779,Y 101.711,Z 77.000,A 180.000,B 0.000,C 180.000} C_DIS
LIN {X 87.865,Y 101.902,Z 77.000,A 180.000,B 0.000,C 180.000} C_DIS
LIN {X 87.946,Y 102.081,Z 77.000,A 180.000,B 0.000,C 180.000} C_DIS
LIN {X 87.958,Y 102.106,Z 77.000,A 180.000,B 0.000,C 180.000} C_DIS
LIN {X 88.037,Y 102.260,Z 77.000,A 180.000,B 0.000,C 180.000} C_DIS
LIN {X 88.137,Y 102.453,Z 77.000,A 180.000,B 0.000,C 180.000} C_DIS
LIN {X 88.224,Y 102.617,Z 77.000,A 180.000,B 0.000,C 180.000} C_DIS
LIN {X 88.316,Y 102.778,Z 77.000,A 180.000,B 0.000,C 180.000} C_DIS
LIN {X 88.494,Y 103.081,Z 77.000,A 180.000,B 0.000,C 180.000} C_DIS
LIN {X 88.539,Y 103.153,Z 77.000,A 180.000,B 0.000,C 180.000} C_DIS
LIN {X 88.657,Y 103.332,Z 77.000,A 180.000,B 0.000,C 180.000} C_DIS
LIN {X 88.777,Y 103.511,Z 77.000,A 180.000,B 0.000,C 180.000} C_DIS
LIN {X 88.852,Y 103.619,Z 77.000,A 180.000,B 0.000,C 180.000} C_DIS
LIN {X 88.903,Y 103.690,Z 77.000,A 180.000,B 0.000,C 180.000} C_DIS
LIN {X 89.031,Y 103.861,Z 77.000,A 180.000,B 0.000,C 180.000} C_DIS
LIN {X 89.171,Y 104.047,Z 77.000,A 180.000,B 0.000,C 180.000} C_DIS
LIN {X 89.209,Y 104.098,Z 77.000,A 180.000,B 0.000,C 180.000} C_DIS
LIN {X 89.315,Y 104.226,Z 77.000,A 180.000,B 0.000,C 180.000} C_DIS
LIN {X 89.466,Y 104.405,Z 77.000,A 180.000,B 0.000,C 180.000} C_DIS
LIN {X 89.567,Y 104.523,Z 77.000,A 180.000,B 0.000,C 180.000} C_DIS
LIN {X 89.623,Y 104.584,Z 77.000,A 180.000,B 0.000,C 180.000} C_DIS
LIN {X 89.746,Y 104.714,Z 77.000,A 180.000,B 0.000,C 180.000} C_DIS
LIN {X 89.960,Y 104.941,Z 77.000,A 180.000,B 0.000,C 180.000} C_DIS
LIN {X 90.103,Y 105.085,Z 77.000,A 180.000,B 0.000,C 180.000} C_DIS
LIN {X 90.330,Y 105.299,Z 77.000,A 180.000,B 0.000,C 180.000} C_DIS
LIN {X 90.461,Y 105.418,Z 77.000,A 180.000,B 0.000,C 180.000} C_DIS
LIN {X 90.531,Y 105.477,Z 77.000,A 180.000,B 0.000,C 180.000} C_DIS
LIN {X 90.743,Y 105.656,Z 77.000,A 180.000,B 0.000,C 180.000} C_DIS
LIN {X 90.818,Y 105.720,Z 77.000,A 180.000,B 0.000,C 180.000} C_DIS
LIN {X 90.960,Y 105.835,Z 77.000,A 180.000,B 0.000,C 180.000} C_DIS
LIN {X 90.997,Y 105.863,Z 77.000,A 180.000,B 0.000,C 180.000} C_DIS
LIN {X 91.197,Y 106.014,Z 77.000,A 180.000,B 0.000,C 180.000} C_DIS
LIN {X 91.355,Y 106.131,Z 77.000,A 180.000,B 0.000,C 180.000} C_DIS
LIN {X 91.444,Y 106.193,Z 77.000,A 180.000,B 0.000,C 180.000} C_DIS
LIN {X 91.712,Y 106.372,Z 77.000,A 180.000,B 0.000,C 180.000} C_DIS
LIN {X 91.891,Y 106.487,Z 77.000,A 180.000,B 0.000,C 180.000} C_DIS
LIN {X 91.994,Y 106.550,Z 77.000,A 180.000,B 0.000,C 180.000} C_DIS
LIN {X 92.297,Y 106.729,Z 77.000,A 180.000,B 0.000,C 180.000} C_DIS
LIN {X 92.427,Y 106.802,Z 77.000,A 180.000,B 0.000,C 180.000} C_DIS
LIN {X 92.632,Y 106.908,Z 77.000,A 180.000,B 0.000,C 180.000} C_DIS
LIN {X 92.785,Y 106.987,Z 77.000,A 180.000,B 0.000,C 180.000} C_DIS
LIN {X 92.964,Y 107.073,Z 77.000,A 180.000,B 0.000,C 180.000} C_DIS
LIN {X 92.993,Y 107.086,Z 77.000,A 180.000,B 0.000,C 180.000} C_DIS
LIN {X 93.142,Y 107.154,Z 77.000,A 180.000,B 0.000,C 180.000} C_DIS
LIN {X 93.391,Y 107.265,Z 77.000,A 180.000,B 0.000,C 180.000} C_DIS
LIN {X 93.500,Y 107.311,Z 77.000,A 180.000,B 0.000,C 180.000} C_DIS
LIN {X 93.679,Y 107.380,Z 77.000,A 180.000,B 0.000,C 180.000} C_DIS
LIN {X 93.857,Y 107.448,Z 77.000,A 180.000,B 0.000,C 180.000} C_DIS
LIN {X 94.036,Y 107.511,Z 77.000,A 180.000,B 0.000,C 180.000} C_DIS
LIN {X 94.215,Y 107.569,Z 77.000,A 180.000,B 0.000,C 180.000} C_DIS
LIN {X 94.394,Y 107.626,Z 77.000,A 180.000,B 0.000,C 180.000} C_DIS
LIN {X 94.573,Y 107.683,Z 77.000,A 180.000,B 0.000,C 180.000} C_DIS
LIN {X 94.751,Y 107.731,Z 77.000,A 180.000,B 0.000,C 180.000} C_DIS
LIN {X 95.026,Y 107.802,Z 77.000,A 180.000,B 0.000,C 180.000} C_DIS
LIN {X 95.109,Y 107.822,Z 77.000,A 180.000,B 0.000,C 180.000} C_DIS
LIN {X 95.288,Y 107.859,Z 77.000,A 180.000,B 0.000,C 180.000} C_DIS
LIN {X 95.466,Y 107.894,Z 77.000,A 180.000,B 0.000,C 180.000} C_DIS
LIN {X 95.645,Y 107.929,Z 77.000,A 180.000,B 0.000,C 180.000} C_DIS
LIN {X 95.824,Y 107.961,Z 77.000,A 180.000,B 0.000,C 180.000} C_DIS
LIN {X 95.959,Y 107.980,Z 77.000,A 180.000,B 0.000,C 180.000} C_DIS
LIN {X 96.181,Y 108.012,Z 77.000,A 180.000,B 0.000,C 180.000} C_DIS
LIN {X 96.360,Y 108.033,Z 77.000,A 180.000,B 0.000,C 180.000} C_DIS
LIN {X 96.539,Y 108.049,Z 77.000,A 180.000,B 0.000,C 180.000} C_DIS
LIN {X 96.718,Y 108.064,Z 77.000,A 180.000,B 0.000,C 180.000} C_DIS
LIN {X 96.897,Y 108.076,Z 77.000,A 180.000,B 0.000,C 180.000} C_DIS
LIN {X 97.075,Y 108.085,Z 77.000,A 180.000,B 0.000,C 180.000} C_DIS
LIN {X 97.433,Y 108.095,Z 77.000,A 180.000,B 0.000,C 180.000} C_DIS
LIN {X 97.612,Y 108.094,Z 77.000,A 180.000,B 0.000,C 180.000} C_DIS
LIN {X 97.969,Y 108.084,Z 77.000,A 180.000,B 0.000,C 180.000} C_DIS
LIN {X 98.148,Y 108.074,Z 77.000,A 180.000,B 0.000,C 180.000} C_DIS
LIN {X 98.327,Y 108.060,Z 77.000,A 180.000,B 0.000,C 180.000} C_DIS
LIN {X 98.505,Y 108.045,Z 77.000,A 180.000,B 0.000,C 180.000} C_DIS
LIN {X 98.684,Y 108.029,Z 77.000,A 180.000,B 0.000,C 180.000} C_DIS
LIN {X 98.863,Y 108.005,Z 77.000,A 180.000,B 0.000,C 180.000} C_DIS
LIN {X 99.042,Y 107.980,Z 77.000,A 180.000,B 0.000,C 180.000} C_DIS
LIN {X 99.221,Y 107.954,Z 77.000,A 180.000,B 0.000,C 180.000} C_DIS
LIN {X 99.399,Y 107.921,Z 77.000,A 180.000,B 0.000,C 180.000} C_DIS
LIN {X 99.578,Y 107.885,Z 77.000,A 180.000,B 0.000,C 180.000} C_DIS
LIN {X 99.757,Y 107.850,Z 77.000,A 180.000,B 0.000,C 180.000} C_DIS
LIN {X 99.936,Y 107.811,Z 77.000,A 180.000,B 0.000,C 180.000} C_DIS
LIN {X 99.974,Y 107.802,Z 77.000,A 180.000,B 0.000,C 180.000} C_DIS
LIN {X 100.293,Y 107.719,Z 77.000,A 180.000,B 0.000,C 180.000} C_DIS
LIN {X 100.472,Y 107.669,Z 77.000,A 180.000,B 0.000,C 180.000} C_DIS
LIN {X 100.829,Y 107.555,Z 77.000,A 180.000,B 0.000,C 180.000} C_DIS
LIN {X 101.008,Y 107.497,Z 77.000,A 180.000,B 0.000,C 180.000} C_DIS
LIN {X 101.153,Y 107.444,Z 77.000,A 180.000,B 0.000,C 180.000} C_DIS
LIN {X 101.366,Y 107.363,Z 77.000,A 180.000,B 0.000,C 180.000} C_DIS
LIN {X 101.545,Y 107.293,Z 77.000,A 180.000,B 0.000,C 180.000} C_DIS
LIN {X 101.609,Y 107.265,Z 77.000,A 180.000,B 0.000,C 180.000} C_DIS
LIN {X 101.902,Y 107.134,Z 77.000,A 180.000,B 0.000,C 180.000} C_DIS
LIN {X 102.007,Y 107.086,Z 77.000,A 180.000,B 0.000,C 180.000} C_DIS
LIN {X 102.081,Y 107.052,Z 77.000,A 180.000,B 0.000,C 180.000} C_DIS
LIN {X 102.260,Y 106.964,Z 77.000,A 180.000,B 0.000,C 180.000} C_DIS
LIN {X 102.438,Y 106.871,Z 77.000,A 180.000,B 0.000,C 180.000} C_DIS
LIN {X 102.617,Y 106.778,Z 77.000,A 180.000,B 0.000,C 180.000} C_DIS
LIN {X 102.703,Y 106.729,Z 77.000,A 180.000,B 0.000,C 180.000} C_DIS
LIN {X 103.006,Y 106.550,Z 77.000,A 180.000,B 0.000,C 180.000} C_DIS
LIN {X 103.153,Y 106.459,Z 77.000,A 180.000,B 0.000,C 180.000} C_DIS
LIN {X 103.288,Y 106.371,Z 77.000,A 180.000,B 0.000,C 180.000} C_DIS
LIN {X 103.556,Y 106.193,Z 77.000,A 180.000,B 0.000,C 180.000} C_DIS
LIN {X 103.690,Y 106.099,Z 77.000,A 180.000,B 0.000,C 180.000} C_DIS
LIN {X 103.803,Y 106.014,Z 77.000,A 180.000,B 0.000,C 180.000} C_DIS
LIN {X 103.869,Y 105.965,Z 77.000,A 180.000,B 0.000,C 180.000} C_DIS
LIN {X 104.040,Y 105.835,Z 77.000,A 180.000,B 0.000,C 180.000} C_DIS
LIN {X 104.047,Y 105.829,Z 77.000,A 180.000,B 0.000,C 180.000} C_DIS
LIN {X 104.226,Y 105.683,Z 77.000,A 180.000,B 0.000,C 180.000} C_DIS
LIN {X 104.414,Y 105.524,Z 77.000,A 180.000,B 0.000,C 180.000} C_DIS
; Link Move Starts
LIN {X 104.632,Y 105.335,Z 77.000,A 180.000,B 0.000,C 180.000} C_DIS
LIN {X 104.860,Y 105.120,Z 76.999,A 180.000,B 0.000,C 180.000} C_DIS
LIN {X 105.066,Y 104.915,Z 76.998,A 180.000,B 0.000,C 180.000} C_DIS
LIN {X 105.283,Y 104.687,Z 76.996,A 180.000,B 0.000,C 180.000} C_DIS
LIN {X 105.486,Y 104.466,Z 76.994,A 180.000,B 0.000,C 180.000} C_DIS
LIN {X 105.681,Y 104.236,Z 76.992,A 180.000,B 0.000,C 180.000} C_DIS
LIN {X 105.864,Y 104.009,Z 76.989,A 180.000,B 0.000,C 180.000} C_DIS
LIN {X 106.051,Y 103.763,Z 76.986,A 180.000,B 0.000,C 180.000} C_DIS
LIN {X 106.226,Y 103.522,Z 76.983,A 180.000,B 0.000,C 180.000} C_DIS
LIN {X 106.401,Y 103.263,Z 76.978,A 180.000,B 0.000,C 180.000} C_DIS
LIN {X 106.556,Y 103.019,Z 76.974,A 180.000,B 0.000,C 180.000} C_DIS
LIN {X 106.718,Y 102.750,Z 76.969,A 180.000,B 0.000,C 180.000} C_DIS
LIN {X 106.862,Y 102.493,Z 76.964,A 180.000,B 0.000,C 180.000} C_DIS
LIN {X 106.934,Y 102.355,Z 76.962,A 180.000,B 0.000,C 180.000} C_DIS
LIN {X 107.007,Y 102.217,Z 76.959,A 180.000,B 0.000,C 180.000} C_DIS
LIN {X 107.073,Y 102.088,Z 76.956,A 180.000,B 0.000,C 180.000} C_DIS
LIN {X 107.135,Y 101.957,Z 76.953,A 180.000,B 0.000,C 180.000} C_DIS
LIN {X 107.199,Y 101.817,Z 76.950,A 180.000,B 0.000,C 180.000} C_DIS
LIN {X 107.263,Y 101.677,Z 76.947,A 180.000,B 0.000,C 180.000} C_DIS
LIN {X 107.322,Y 101.539,Z 76.944,A 180.000,B 0.000,C 180.000} C_DIS
LIN {X 107.378,Y 101.399,Z 76.941,A 180.000,B 0.000,C 180.000} C_DIS
LIN {X 107.435,Y 101.254,Z 76.937,A 180.000,B 0.000,C 180.000} C_DIS
LIN {X 107.492,Y 101.110,Z 76.934,A 180.000,B 0.000,C 180.000} C_DIS
LIN {X 107.544,Y 100.974,Z 76.930,A 180.000,B 0.000,C 180.000} C_DIS
LIN {X 107.591,Y 100.836,Z 76.927,A 180.000,B 0.000,C 180.000} C_DIS
LIN {X 107.640,Y 100.686,Z 76.923,A 180.000,B 0.000,C 180.000} C_DIS
LIN {X 107.690,Y 100.537,Z 76.919,A 180.000,B 0.000,C 180.000} C_DIS
LIN {X 107.731,Y 100.397,Z 76.915,A 180.000,B 0.000,C 180.000} C_DIS
LIN {X 107.769,Y 100.257,Z 76.911,A 180.000,B 0.000,C 180.000} C_DIS
LIN {X 107.810,Y 100.106,Z 76.907,A 180.000,B 0.000,C 180.000} C_DIS
LIN {X 107.851,Y 99.955,Z 76.903,A 180.000,B 0.000,C 180.000} C_DIS
LIN {X 107.888,Y 99.813,Z 76.899,A 180.000,B 0.000,C 180.000} C_DIS
LIN {X 107.919,Y 99.669,Z 76.895,A 180.000,B 0.000,C 180.000} C_DIS
LIN {X 107.951,Y 99.516,Z 76.891,A 180.000,B 0.000,C 180.000} C_DIS
LIN {X 107.984,Y 99.362,Z 76.886,A 180.000,B 0.000,C 180.000} C_DIS
LIN {X 108.010,Y 99.218,Z 76.882,A 180.000,B 0.000,C 180.000} C_DIS
LIN {X 108.032,Y 99.073,Z 76.878,A 180.000,B 0.000,C 180.000} C_DIS
LIN {X 108.056,Y 98.921,Z 76.873,A 180.000,B 0.000,C 180.000} C_DIS
LIN {X 108.079,Y 98.768,Z 76.868,A 180.000,B 0.000,C 180.000} C_DIS
LIN {X 108.099,Y 98.620,Z 76.864,A 180.000,B 0.000,C 180.000} C_DIS
LIN {X 108.114,Y 98.471,Z 76.859,A 180.000,B 0.000,C 180.000} C_DIS
LIN {X 108.130,Y 98.315,Z 76.854,A 180.000,B 0.000,C 180.000} C_DIS
LIN {X 108.145,Y 98.159,Z 76.849,A 180.000,B 0.000,C 180.000} C_DIS
LIN {X 108.155,Y 98.012,Z 76.844,A 180.000,B 0.000,C 180.000} C_DIS
LIN {X 108.164,Y 97.789,Z 76.837,A 180.000,B 0.000,C 180.000} C_DIS
LIN {X 108.168,Y 97.713,Z 76.835,A 180.000,B 0.000,C 180.000} C_DIS
LIN {X 108.171,Y 97.637,Z 76.832,A 180.000,B 0.000,C 180.000} C_DIS
LIN {X 108.173,Y 97.561,Z 76.829,A 180.000,B 0.000,C 180.000} C_DIS
LIN {X 108.174,Y 97.485,Z 76.827,A 180.000,B 0.000,C 180.000} C_DIS
LIN {X 108.175,Y 97.409,Z 76.824,A 180.000,B 0.000,C 180.000} C_DIS
LIN {X 108.175,Y 97.333,Z 76.822,A 180.000,B 0.000,C 180.000} C_DIS
LIN {X 108.173,Y 97.179,Z 76.816,A 180.000,B 0.000,C 180.000} C_DIS
LIN {X 108.172,Y 97.100,Z 76.814,A 180.000,B 0.000,C 180.000} C_DIS
LIN {X 108.171,Y 97.022,Z 76.811,A 180.000,B 0.000,C 180.000} C_DIS
LIN {X 108.170,Y 96.943,Z 76.808,A 180.000,B 0.000,C 180.000} C_DIS
LIN {X 108.168,Y 96.870,Z 76.806,A 180.000,B 0.000,C 180.000} C_DIS
LIN {X 108.163,Y 96.796,Z 76.803,A 180.000,B 0.000,C 180.000} C_DIS
LIN {X 108.148,Y 96.574,Z 76.795,A 180.000,B 0.000,C 180.000} C_DIS
LIN {X 108.138,Y 96.423,Z 76.790,A 180.000,B 0.000,C 180.000} C_DIS
LIN {X 108.131,Y 96.347,Z 76.787,A 180.000,B 0.000,C 180.000} C_DIS
LIN {X 108.123,Y 96.271,Z 76.785,A 180.000,B 0.000,C 180.000} C_DIS
LIN {X 108.115,Y 96.195,Z 76.782,A 180.000,B 0.000,C 180.000} C_DIS
LIN {X 108.106,Y 96.118,Z 76.779,A 180.000,B 0.000,C 180.000} C_DIS
LIN {X 108.096,Y 96.042,Z 76.777,A 180.000,B 0.000,C 180.000} C_DIS
LIN {X 108.077,Y 95.887,Z 76.771,A 180.000,B 0.000,C 180.000} C_DIS
LIN {X 108.067,Y 95.809,Z 76.768,A 180.000,B 0.000,C 180.000} C_DIS
LIN {X 108.057,Y 95.731,Z 76.766,A 180.000,B 0.000,C 180.000} C_DIS
LIN {X 108.046,Y 95.658,Z 76.763,A 180.000,B 0.000,C 180.000} C_DIS
LIN {X 108.033,Y 95.585,Z 76.761,A 180.000,B 0.000,C 180.000} C_DIS
LIN {X 107.993,Y 95.365,Z 76.753,A 180.000,B 0.000,C 180.000} C_DIS
LIN {X 107.966,Y 95.218,Z 76.748,A 180.000,B 0.000,C 180.000} C_DIS
LIN {X 107.952,Y 95.144,Z 76.745,A 180.000,B 0.000,C 180.000} C_DIS
LIN {X 107.934,Y 95.068,Z 76.742,A 180.000,B 0.000,C 180.000} C_DIS
LIN {X 107.916,Y 94.993,Z 76.739,A 180.000,B 0.000,C 180.000} C_DIS
LIN {X 107.898,Y 94.917,Z 76.737,A 180.000,B 0.000,C 180.000} C_DIS
LIN {X 107.880,Y 94.842,Z 76.734,A 180.000,B 0.000,C 180.000} C_DIS
LIN {X 107.843,Y 94.690,Z 76.729,A 180.000,B 0.000,C 180.000} C_DIS
LIN {X 107.825,Y 94.614,Z 76.726,A 180.000,B 0.000,C 180.000} C_DIS
LIN {X 107.807,Y 94.538,Z 76.723,A 180.000,B 0.000,C 180.000} C_DIS
LIN {X 107.787,Y 94.466,Z 76.721,A 180.000,B 0.000,C 180.000} C_DIS
LIN {X 107.766,Y 94.395,Z 76.718,A 180.000,B 0.000,C 180.000} C_DIS
LIN {X 107.680,Y 94.108,Z 76.707,A 180.000,B 0.000,C 180.000} C_DIS
LIN {X 107.658,Y 94.036,Z 76.705,A 180.000,B 0.000,C 180.000} C_DIS
LIN {X 107.635,Y 93.965,Z 76.702,A 180.000,B 0.000,C 180.000} C_DIS
LIN {X 107.609,Y 93.891,Z 76.700,A 180.000,B 0.000,C 180.000} C_DIS
LIN {X 107.556,Y 93.745,Z 76.694,A 180.000,B 0.000,C 180.000} C_DIS
LIN {X 107.530,Y 93.671,Z 76.691,A 180.000,B 0.000,C 180.000} C_DIS
LIN {X 107.477,Y 93.528,Z 76.686,A 180.000,B 0.000,C 180.000} C_DIS
LIN {X 107.450,Y 93.456,Z 76.683,A 180.000,B 0.000,C 180.000} C_DIS
LIN {X 107.423,Y 93.384,Z 76.681,A 180.000,B 0.000,C 180.000} C_DIS
LIN {X 107.395,Y 93.313,Z 76.678,A 180.000,B 0.000,C 180.000} C_DIS
LIN {X 107.366,Y 93.243,Z 76.675,A 180.000,B 0.000,C 180.000} C_DIS
LIN {X 107.245,Y 92.960,Z 76.665,A 180.000,B 0.000,C 180.000} C_DIS
LIN {X 107.214,Y 92.889,Z 76.662,A 180.000,B 0.000,C 180.000} C_DIS
LIN {X 107.182,Y 92.819,Z 76.659,A 180.000,B 0.000,C 180.000} C_DIS
LIN {X 107.149,Y 92.751,Z 76.657,A 180.000,B 0.000,C 180.000} C_DIS
LIN {X 107.013,Y 92.477,Z 76.646,A 180.000,B 0.000,C 180.000} C_DIS
LIN {X 106.979,Y 92.408,Z 76.643,A 180.000,B 0.000,C 180.000} C_DIS
LIN {X 106.944,Y 92.340,Z 76.640,A 180.000,B 0.000,C 180.000} C_DIS
LIN {X 106.908,Y 92.272,Z 76.638,A 180.000,B 0.000,C 180.000} C_DIS
LIN {X 106.872,Y 92.205,Z 76.635,A 180.000,B 0.000,C 180.000} C_DIS
LIN {X 106.834,Y 92.138,Z 76.632,A 180.000,B 0.000,C 180.000} C_DIS
LIN {X 106.683,Y 91.872,Z 76.622,A 180.000,B 0.000,C 180.000} C_DIS
LIN {X 106.645,Y 91.805,Z 76.619,A 180.000,B 0.000,C 180.000} C_DIS
LIN {X 106.605,Y 91.740,Z 76.616,A 180.000,B 0.000,C 180.000} C_DIS
LIN {X 106.564,Y 91.675,Z 76.614,A 180.000,B 0.000,C 180.000} C_DIS
LIN {X 106.398,Y 91.417,Z 76.603,A 180.000,B 0.000,C 180.000} C_DIS
LIN {X 106.357,Y 91.353,Z 76.600,A 180.000,B 0.000,C 180.000} C_DIS
LIN {X 106.314,Y 91.290,Z 76.598,A 180.000,B 0.000,C 180.000} C_DIS
LIN {X 106.270,Y 91.228,Z 76.595,A 180.000,B 0.000,C 180.000} C_DIS
LIN {X 106.226,Y 91.165,Z 76.592,A 180.000,B 0.000,C 180.000} C_DIS
LIN {X 106.180,Y 91.102,Z 76.590,A 180.000,B 0.000,C 180.000} C_DIS
LIN {X 106.000,Y 90.853,Z 76.579,A 180.000,B 0.000,C 180.000} C_DIS
LIN {X 105.955,Y 90.792,Z 76.576,A 180.000,B 0.000,C 180.000} C_DIS
LIN {X 105.908,Y 90.731,Z 76.574,A 180.000,B 0.000,C 180.000} C_DIS
LIN {X 105.860,Y 90.671,Z 76.571,A 180.000,B 0.000,C 180.000} C_DIS
LIN {X 105.664,Y 90.432,Z 76.560,A 180.000,B 0.000,C 180.000} C_DIS
LIN {X 105.617,Y 90.374,Z 76.557,A 180.000,B 0.000,C 180.000} C_DIS
LIN {X 105.568,Y 90.316,Z 76.555,A 180.000,B 0.000,C 180.000} C_DIS
LIN {X 105.517,Y 90.260,Z 76.552,A 180.000,B 0.000,C 180.000} C_DIS
LIN {X 105.465,Y 90.202,Z 76.549,A 180.000,B 0.000,C 180.000} C_DIS
LIN {X 105.412,Y 90.144,Z 76.547,A 180.000,B 0.000,C 180.000} C_DIS
LIN {X 105.203,Y 89.917,Z 76.536,A 180.000,B 0.000,C 180.000} C_DIS
LIN {X 105.152,Y 89.861,Z 76.533,A 180.000,B 0.000,C 180.000} C_DIS
LIN {X 105.099,Y 89.806,Z 76.531,A 180.000,B 0.000,C 180.000} C_DIS
LIN {X 105.044,Y 89.751,Z 76.528,A 180.000,B 0.000,C 180.000} C_DIS
LIN {X 104.822,Y 89.535,Z 76.517,A 180.000,B 0.000,C 180.000} C_DIS
LIN {X 104.768,Y 89.482,Z 76.514,A 180.000,B 0.000,C 180.000} C_DIS
LIN {X 104.712,Y 89.431,Z 76.512,A 180.000,B 0.000,C 180.000} C_DIS
LIN {X 104.656,Y 89.381,Z 76.509,A 180.000,B 0.000,C 180.000} C_DIS
LIN {X 104.419,Y 89.174,Z 76.498,A 180.000,B 0.000,C 180.000} C_DIS
LIN {X 104.362,Y 89.124,Z 76.496,A 180.000,B 0.000,C 180.000} C_DIS
LIN {X 104.304,Y 89.074,Z 76.493,A 180.000,B 0.000,C 180.000} C_DIS
LIN {X 104.245,Y 89.025,Z 76.490,A 180.000,B 0.000,C 180.000} C_DIS
LIN {X 104.186,Y 88.976,Z 76.488,A 180.000,B 0.000,C 180.000} C_DIS
LIN {X 104.125,Y 88.928,Z 76.485,A 180.000,B 0.000,C 180.000} C_DIS
LIN {X 103.880,Y 88.737,Z 76.474,A 180.000,B 0.000,C 180.000} C_DIS
LIN {X 103.820,Y 88.691,Z 76.471,A 180.000,B 0.000,C 180.000} C_DIS
LIN {X 103.760,Y 88.646,Z 76.469,A 180.000,B 0.000,C 180.000} C_DIS
LIN {X 103.697,Y 88.603,Z 76.466,A 180.000,B 0.000,C 180.000} C_DIS
LIN {X 103.438,Y 88.423,Z 76.455,A 180.000,B 0.000,C 180.000} C_DIS
LIN {X 103.376,Y 88.380,Z 76.452,A 180.000,B 0.000,C 180.000} C_DIS
LIN {X 103.313,Y 88.338,Z 76.450,A 180.000,B 0.000,C 180.000} C_DIS
LIN {X 103.249,Y 88.296,Z 76.447,A 180.000,B 0.000,C 180.000} C_DIS
LIN {X 103.185,Y 88.255,Z 76.444,A 180.000,B 0.000,C 180.000} C_DIS
LIN {X 103.118,Y 88.214,Z 76.442,A 180.000,B 0.000,C 180.000} C_DIS
LIN {X 102.852,Y 88.051,Z 76.431,A 180.000,B 0.000,C 180.000} C_DIS
LIN {X 102.788,Y 88.012,Z 76.428,A 180.000,B 0.000,C 180.000} C_DIS
LIN {X 102.722,Y 87.974,Z 76.426,A 180.000,B 0.000,C 180.000} C_DIS
LIN {X 102.655,Y 87.938,Z 76.423,A 180.000,B 0.000,C 180.000} C_DIS
LIN {X 102.377,Y 87.789,Z 76.412,A 180.000,B 0.000,C 180.000} C_DIS
LIN {X 102.310,Y 87.752,Z 76.409,A 180.000,B 0.000,C 180.000} C_DIS
LIN {X 102.242,Y 87.718,Z 76.407,A 180.000,B 0.000,C 180.000} C_DIS
LIN {X 102.173,Y 87.684,Z 76.404,A 180.000,B 0.000,C 180.000} C_DIS
LIN {X 102.104,Y 87.651,Z 76.401,A 180.000,B 0.000,C 180.000} C_DIS
LIN {X 102.034,Y 87.617,Z 76.398,A 180.000,B 0.000,C 180.000} C_DIS
